// TIA Portal V19 export
FUNCTION "AUTO_LOGIC_FOR_CIP_TANK" : Void   // FC13, LAD
{ S7_Optimized_Access := 'TRUE' }
// stored: SetENOAutomatically false
   VAR_TEMP   // added for the SCL form of the ladder/FBD networks
      _w1 : Bool;
      _w2 : Bool;
      _w3 : Bool;
      _w4 : Bool;
   END_VAR
BEGIN

REGION Network 1: START
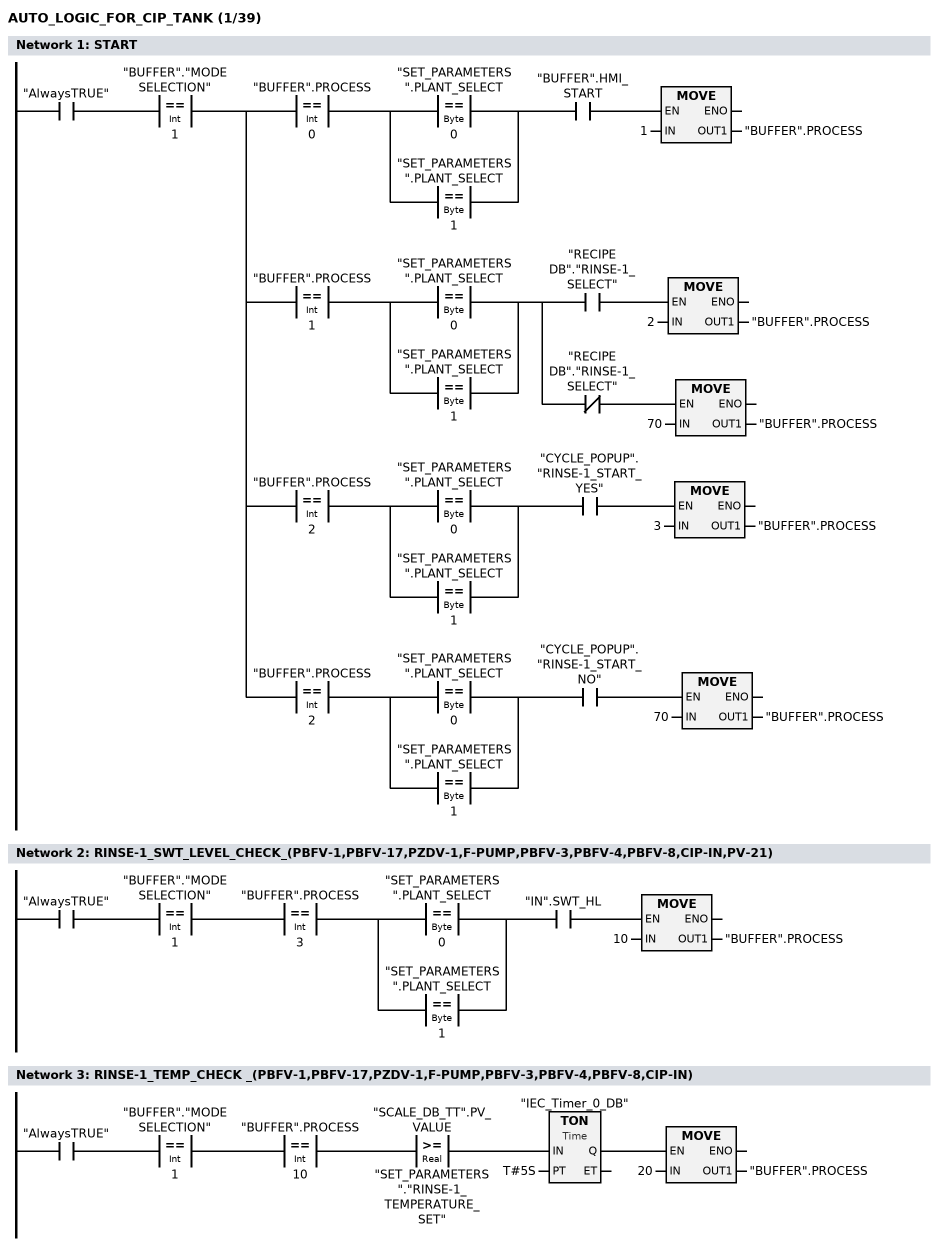
   RUNG wire#powerrail
      Contact( "AlwaysTRUE" )
      { S7_Templates := "SrcType := Int" } EQ_Contact(in1 := "BUFFER"."MODE SELECTION", in2 := 1)
      wire#w1
      { S7_Templates := "SrcType := Int" } EQ_Contact(in1 := "BUFFER".PROCESS, in2 := 0)
      wire#w2
      { S7_Templates := "SrcType := Byte" } EQ_Contact(in1 := "SET_PARAMETERS".PLANT_SELECT, in2 := 0)
      wire#w3
      Contact( "BUFFER".HMI_START )
      Move(in := 1, out1 => "BUFFER".PROCESS)
   END_RUNG
   RUNG wire#w2
      { S7_Templates := "SrcType := Byte" } EQ_Contact(in1 := "SET_PARAMETERS".PLANT_SELECT, in2 := 1)
   END_RUNG wire#w3
   RUNG wire#w1
      { S7_Templates := "SrcType := Int" } EQ_Contact(in1 := "BUFFER".PROCESS, in2 := 1)
      wire#w4
      { S7_Templates := "SrcType := Byte" } EQ_Contact(in1 := "SET_PARAMETERS".PLANT_SELECT, in2 := 0)
      wire#w5
      Contact( "RECIPE DB"."RINSE-1_SELECT" )
      Move(in := 2, out1 => "BUFFER".PROCESS)
   END_RUNG
   RUNG wire#w4
      { S7_Templates := "SrcType := Byte" } EQ_Contact(in1 := "SET_PARAMETERS".PLANT_SELECT, in2 := 1)
   END_RUNG wire#w5
   RUNG wire#w5
      I_Contact( "RECIPE DB"."RINSE-1_SELECT" )
      Move(in := 70, out1 => "BUFFER".PROCESS)
   END_RUNG
   RUNG wire#w1
      { S7_Templates := "SrcType := Int" } EQ_Contact(in1 := "BUFFER".PROCESS, in2 := 2)
      wire#w6
      { S7_Templates := "SrcType := Byte" } EQ_Contact(in1 := "SET_PARAMETERS".PLANT_SELECT, in2 := 0)
      wire#w7
      Contact( "CYCLE_POPUP"."RINSE-1_START_YES" )
      Move(in := 3, out1 => "BUFFER".PROCESS)
   END_RUNG
   RUNG wire#w6
      { S7_Templates := "SrcType := Byte" } EQ_Contact(in1 := "SET_PARAMETERS".PLANT_SELECT, in2 := 1)
   END_RUNG wire#w7
   RUNG wire#w1
      { S7_Templates := "SrcType := Int" } EQ_Contact(in1 := "BUFFER".PROCESS, in2 := 2)
      wire#w8
      { S7_Templates := "SrcType := Byte" } EQ_Contact(in1 := "SET_PARAMETERS".PLANT_SELECT, in2 := 0)
      wire#w9
      Contact( "CYCLE_POPUP"."RINSE-1_START_NO" )
      Move(in := 70, out1 => "BUFFER".PROCESS)
   END_RUNG
   RUNG wire#w8
      { S7_Templates := "SrcType := Byte" } EQ_Contact(in1 := "SET_PARAMETERS".PLANT_SELECT, in2 := 1)
   END_RUNG wire#w9
   // the same network as SCL:
   #_w1 := "AlwaysTRUE" AND ("BUFFER"."MODE SELECTION" = 1);
   IF #_w1 AND ("BUFFER".PROCESS = 0) AND (("SET_PARAMETERS".PLANT_SELECT = 0) OR ("SET_PARAMETERS".PLANT_SELECT = 1)) AND "BUFFER".HMI_START THEN
       "BUFFER".PROCESS := 1;
   END_IF;
   #_w2 := #_w1 AND ("BUFFER".PROCESS = 1) AND (("SET_PARAMETERS".PLANT_SELECT = 0) OR ("SET_PARAMETERS".PLANT_SELECT = 1));
   IF #_w2 AND "RECIPE DB"."RINSE-1_SELECT" THEN "BUFFER".PROCESS := 2; END_IF;
   IF #_w2 AND NOT "RECIPE DB"."RINSE-1_SELECT" THEN "BUFFER".PROCESS := 70; END_IF;
   IF #_w1 AND ("BUFFER".PROCESS = 2) AND (("SET_PARAMETERS".PLANT_SELECT = 0) OR ("SET_PARAMETERS".PLANT_SELECT = 1)) AND "CYCLE_POPUP"."RINSE-1_START_YES" THEN
       "BUFFER".PROCESS := 3;
   END_IF;
   IF #_w1 AND ("BUFFER".PROCESS = 2) AND (("SET_PARAMETERS".PLANT_SELECT = 0) OR ("SET_PARAMETERS".PLANT_SELECT = 1)) AND "CYCLE_POPUP"."RINSE-1_START_NO" THEN
       "BUFFER".PROCESS := 70;
   END_IF;
END_REGION

REGION Network 2: RINSE-1_SWT_LEVEL_CHECK_(PBFV-1,PBFV-17,PZDV-1,F-PUMP,PBFV-3,PBFV-4,PBFV-8,CIP-IN,PV-21)
   RUNG wire#powerrail
      Contact( "AlwaysTRUE" )
      { S7_Templates := "SrcType := Int" } EQ_Contact(in1 := "BUFFER"."MODE SELECTION", in2 := 1)
      { S7_Templates := "SrcType := Int" } EQ_Contact(in1 := "BUFFER".PROCESS, in2 := 3)
      wire#w1
      { S7_Templates := "SrcType := Byte" } EQ_Contact(in1 := "SET_PARAMETERS".PLANT_SELECT, in2 := 0)
      wire#w2
      Contact( "IN".SWT_HL )
      Move(in := 10, out1 => "BUFFER".PROCESS)
   END_RUNG
   RUNG wire#w1
      { S7_Templates := "SrcType := Byte" } EQ_Contact(in1 := "SET_PARAMETERS".PLANT_SELECT, in2 := 1)
   END_RUNG wire#w2
   // the same network as SCL:
   IF "AlwaysTRUE" AND ("BUFFER"."MODE SELECTION" = 1) AND ("BUFFER".PROCESS = 3) AND (("SET_PARAMETERS".PLANT_SELECT = 0) OR ("SET_PARAMETERS".PLANT_SELECT = 1)) AND "IN".SWT_HL THEN
       "BUFFER".PROCESS := 10;
   END_IF;
END_REGION

REGION Network 3: RINSE-1_TEMP_CHECK _(PBFV-1,PBFV-17,PZDV-1,F-PUMP,PBFV-3,PBFV-4,PBFV-8,CIP-IN)
   RUNG wire#powerrail
      Contact( "AlwaysTRUE" )
      { S7_Templates := "SrcType := Int" } EQ_Contact(in1 := "BUFFER"."MODE SELECTION", in2 := 1)
      { S7_Templates := "SrcType := Int" } EQ_Contact(in1 := "BUFFER".PROCESS, in2 := 10)
      { S7_Templates := "SrcType := Real" } GE_Contact(in1 := "SCALE_DB_TT".PV_VALUE, in2 := "SET_PARAMETERS"."RINSE-1_TEMPERATURE_SET")
      { S7_Templates := "time_type := Time" } "IEC_Timer_0_DB".TON(pt := T#5S, et =>)
      Move(in := 20, out1 => "BUFFER".PROCESS)
   END_RUNG
   // the same network as SCL:
   "IEC_Timer_0_DB".TON(IN := "AlwaysTRUE" AND ("BUFFER"."MODE SELECTION" = 1) AND ("BUFFER".PROCESS = 10) AND ("SCALE_DB_TT".PV_VALUE >= "SET_PARAMETERS"."RINSE-1_TEMPERATURE_SET"),
                        PT := T#5S);
   IF "IEC_Timer_0_DB".Q THEN "BUFFER".PROCESS := 20; END_IF;
END_REGION

REGION Network 4: RINSE-1_CLEANING_TIME_(PBFV-1,PBFV-17,PZDV-1,F-PUMP,PBFV-3,PBFV-4,PBFV-8,CIP-IN)
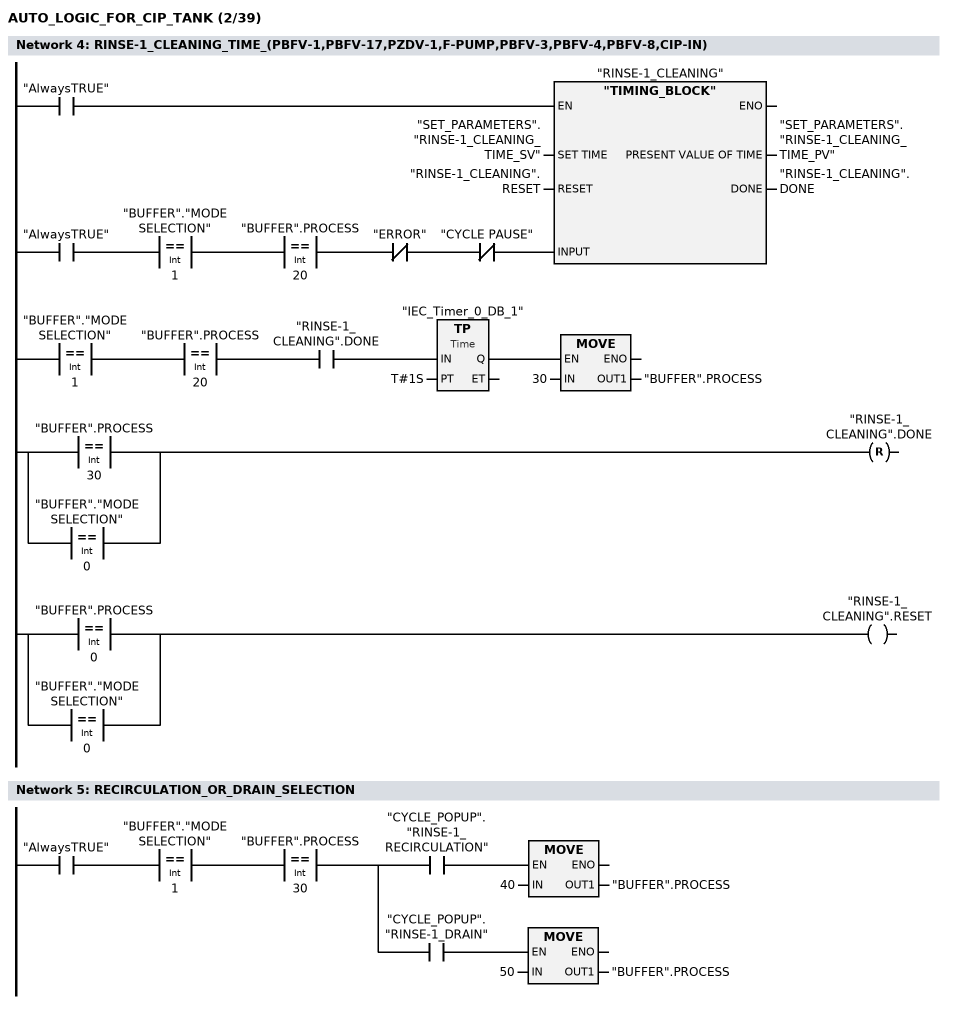
   RUNG wire#powerrail
      Contact( "AlwaysTRUE" )
      "RINSE-1_CLEANING"(INPUT := wire#w1, "SET TIME" := "SET_PARAMETERS"."RINSE-1_CLEANING_TIME_SV", RESET := "RINSE-1_CLEANING".RESET, "PRESENT VALUE OF TIME" => "SET_PARAMETERS"."RINSE-1_CLEANING_TIME_PV", DONE => "RINSE-1_CLEANING".DONE)
   END_RUNG
   RUNG wire#powerrail
      Contact( "AlwaysTRUE" )
      { S7_Templates := "SrcType := Int" } EQ_Contact(in1 := "BUFFER"."MODE SELECTION", in2 := 1)
      { S7_Templates := "SrcType := Int" } EQ_Contact(in1 := "BUFFER".PROCESS, in2 := 20)
      I_Contact( "ERROR" )
      I_Contact( "CYCLE PAUSE" )
   END_RUNG wire#w1
   RUNG wire#powerrail
      { S7_Templates := "SrcType := Int" } EQ_Contact(in1 := "BUFFER"."MODE SELECTION", in2 := 1)
      { S7_Templates := "SrcType := Int" } EQ_Contact(in1 := "BUFFER".PROCESS, in2 := 20)
      Contact( "RINSE-1_CLEANING".DONE )
      { S7_Templates := "time_type := Time" } "IEC_Timer_0_DB_1".TP(pt := T#1S, et =>)
      Move(in := 30, out1 => "BUFFER".PROCESS)
   END_RUNG
   RUNG wire#powerrail
      { S7_Templates := "SrcType := Int" } EQ_Contact(in1 := "BUFFER".PROCESS, in2 := 30)
      wire#w2
      R_Coil( "RINSE-1_CLEANING".DONE )
   END_RUNG
   RUNG wire#powerrail
      { S7_Templates := "SrcType := Int" } EQ_Contact(in1 := "BUFFER"."MODE SELECTION", in2 := 0)
   END_RUNG wire#w2
   RUNG wire#powerrail
      { S7_Templates := "SrcType := Int" } EQ_Contact(in1 := "BUFFER".PROCESS, in2 := 0)
      wire#w3
      Coil( "RINSE-1_CLEANING".RESET )
   END_RUNG
   RUNG wire#powerrail
      { S7_Templates := "SrcType := Int" } EQ_Contact(in1 := "BUFFER"."MODE SELECTION", in2 := 0)
   END_RUNG wire#w3
   // the same network as SCL:
   IF "AlwaysTRUE" THEN
       "RINSE-1_CLEANING"("SET TIME" := "SET_PARAMETERS"."RINSE-1_CLEANING_TIME_SV",   // "TIMING_BLOCK"
                          RESET := "RINSE-1_CLEANING".RESET,
                          INPUT := "AlwaysTRUE" AND ("BUFFER"."MODE SELECTION" = 1) AND ("BUFFER".PROCESS = 20) AND NOT "ERROR" AND NOT "CYCLE PAUSE",
                          "PRESENT VALUE OF TIME" => "SET_PARAMETERS"."RINSE-1_CLEANING_TIME_PV",
                          DONE => "RINSE-1_CLEANING".DONE);
   END_IF;
   "IEC_Timer_0_DB_1".TP(IN := ("BUFFER"."MODE SELECTION" = 1) AND ("BUFFER".PROCESS = 20) AND "RINSE-1_CLEANING".DONE,
                         PT := T#1S);
   IF "IEC_Timer_0_DB_1".Q THEN "BUFFER".PROCESS := 30; END_IF;
   IF ("BUFFER".PROCESS = 30) OR ("BUFFER"."MODE SELECTION" = 0) THEN
       "RINSE-1_CLEANING".DONE := FALSE;
   END_IF;
   "RINSE-1_CLEANING".RESET := ("BUFFER".PROCESS = 0) OR ("BUFFER"."MODE SELECTION" = 0);
END_REGION

REGION Network 5: RECIRCULATION_OR_DRAIN_SELECTION
   RUNG wire#powerrail
      Contact( "AlwaysTRUE" )
      { S7_Templates := "SrcType := Int" } EQ_Contact(in1 := "BUFFER"."MODE SELECTION", in2 := 1)
      { S7_Templates := "SrcType := Int" } EQ_Contact(in1 := "BUFFER".PROCESS, in2 := 30)
      wire#w1
      Contact( "CYCLE_POPUP"."RINSE-1_RECIRCULATION" )
      Move(in := 40, out1 => "BUFFER".PROCESS)
   END_RUNG
   RUNG wire#w1
      Contact( "CYCLE_POPUP"."RINSE-1_DRAIN" )
      Move(in := 50, out1 => "BUFFER".PROCESS)
   END_RUNG
   // the same network as SCL:
   #_w1 := "AlwaysTRUE" AND ("BUFFER"."MODE SELECTION" = 1) AND ("BUFFER".PROCESS = 30);
   IF #_w1 AND "CYCLE_POPUP"."RINSE-1_RECIRCULATION" THEN "BUFFER".PROCESS := 40; END_IF;
   IF #_w1 AND "CYCLE_POPUP"."RINSE-1_DRAIN" THEN "BUFFER".PROCESS := 50; END_IF;
END_REGION

REGION Network 6: RINSE-1_RECIRCULATION_TIME_(CIP-OUT,R-PUMP,PBFV-6,PBFV-8,CIP-IN)
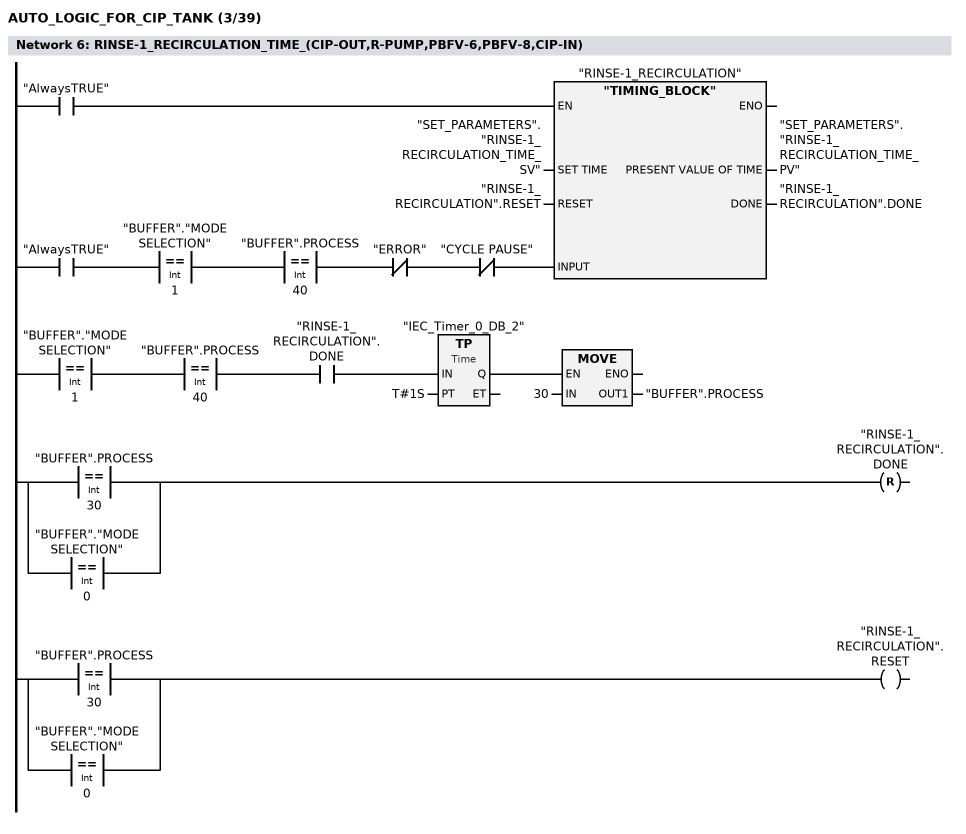
   RUNG wire#powerrail
      Contact( "AlwaysTRUE" )
      "RINSE-1_RECIRCULATION"(INPUT := wire#w1, "SET TIME" := "SET_PARAMETERS"."RINSE-1_RECIRCULATION_TIME_SV", RESET := "RINSE-1_RECIRCULATION".RESET, "PRESENT VALUE OF TIME" => "SET_PARAMETERS"."RINSE-1_RECIRCULATION_TIME_PV", DONE => "RINSE-1_RECIRCULATION".DONE)
   END_RUNG
   RUNG wire#powerrail
      Contact( "AlwaysTRUE" )
      { S7_Templates := "SrcType := Int" } EQ_Contact(in1 := "BUFFER"."MODE SELECTION", in2 := 1)
      { S7_Templates := "SrcType := Int" } EQ_Contact(in1 := "BUFFER".PROCESS, in2 := 40)
      I_Contact( "ERROR" )
      I_Contact( "CYCLE PAUSE" )
   END_RUNG wire#w1
   RUNG wire#powerrail
      { S7_Templates := "SrcType := Int" } EQ_Contact(in1 := "BUFFER"."MODE SELECTION", in2 := 1)
      { S7_Templates := "SrcType := Int" } EQ_Contact(in1 := "BUFFER".PROCESS, in2 := 40)
      Contact( "RINSE-1_RECIRCULATION".DONE )
      { S7_Templates := "time_type := Time" } "IEC_Timer_0_DB_2".TP(pt := T#1S, et =>)
      Move(in := 30, out1 => "BUFFER".PROCESS)
   END_RUNG
   RUNG wire#powerrail
      { S7_Templates := "SrcType := Int" } EQ_Contact(in1 := "BUFFER".PROCESS, in2 := 30)
      wire#w2
      R_Coil( "RINSE-1_RECIRCULATION".DONE )
   END_RUNG
   RUNG wire#powerrail
      { S7_Templates := "SrcType := Int" } EQ_Contact(in1 := "BUFFER"."MODE SELECTION", in2 := 0)
   END_RUNG wire#w2
   RUNG wire#powerrail
      { S7_Templates := "SrcType := Int" } EQ_Contact(in1 := "BUFFER".PROCESS, in2 := 30)
      wire#w3
      Coil( "RINSE-1_RECIRCULATION".RESET )
   END_RUNG
   RUNG wire#powerrail
      { S7_Templates := "SrcType := Int" } EQ_Contact(in1 := "BUFFER"."MODE SELECTION", in2 := 0)
   END_RUNG wire#w3
   // the same network as SCL:
   IF "AlwaysTRUE" THEN
       "RINSE-1_RECIRCULATION"("SET TIME" := "SET_PARAMETERS"."RINSE-1_RECIRCULATION_TIME_SV",   // "TIMING_BLOCK"
                               RESET := "RINSE-1_RECIRCULATION".RESET,
                               INPUT := "AlwaysTRUE" AND ("BUFFER"."MODE SELECTION" = 1) AND ("BUFFER".PROCESS = 40) AND NOT "ERROR" AND NOT "CYCLE PAUSE",
                               "PRESENT VALUE OF TIME" => "SET_PARAMETERS"."RINSE-1_RECIRCULATION_TIME_PV",
                               DONE => "RINSE-1_RECIRCULATION".DONE);
   END_IF;
   "IEC_Timer_0_DB_2".TP(IN := ("BUFFER"."MODE SELECTION" = 1) AND ("BUFFER".PROCESS = 40) AND "RINSE-1_RECIRCULATION".DONE,
                         PT := T#1S);
   IF "IEC_Timer_0_DB_2".Q THEN "BUFFER".PROCESS := 30; END_IF;
   IF ("BUFFER".PROCESS = 30) OR ("BUFFER"."MODE SELECTION" = 0) THEN
       "RINSE-1_RECIRCULATION".DONE := FALSE;
   END_IF;
   "RINSE-1_RECIRCULATION".RESET := ("BUFFER".PROCESS = 30) OR ("BUFFER"."MODE SELECTION" = 0);
END_REGION

REGION Network 7: RINSE-1_DRAIN_TIME_(CIP-OUT,R_PUMP,PBFV-11)
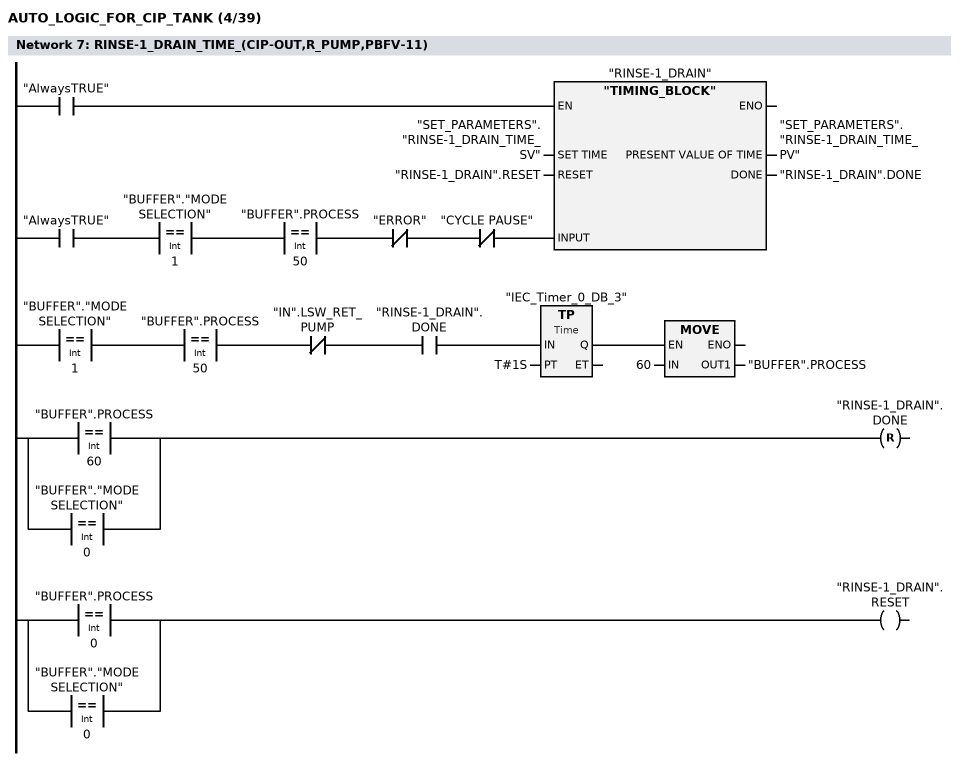
   RUNG wire#powerrail
      Contact( "AlwaysTRUE" )
      "RINSE-1_DRAIN"(INPUT := wire#w1, "SET TIME" := "SET_PARAMETERS"."RINSE-1_DRAIN_TIME_SV", RESET := "RINSE-1_DRAIN".RESET, "PRESENT VALUE OF TIME" => "SET_PARAMETERS"."RINSE-1_DRAIN_TIME_PV", DONE => "RINSE-1_DRAIN".DONE)
   END_RUNG
   RUNG wire#powerrail
      Contact( "AlwaysTRUE" )
      { S7_Templates := "SrcType := Int" } EQ_Contact(in1 := "BUFFER"."MODE SELECTION", in2 := 1)
      { S7_Templates := "SrcType := Int" } EQ_Contact(in1 := "BUFFER".PROCESS, in2 := 50)
      I_Contact( "ERROR" )
      I_Contact( "CYCLE PAUSE" )
   END_RUNG wire#w1
   RUNG wire#powerrail
      { S7_Templates := "SrcType := Int" } EQ_Contact(in1 := "BUFFER"."MODE SELECTION", in2 := 1)
      { S7_Templates := "SrcType := Int" } EQ_Contact(in1 := "BUFFER".PROCESS, in2 := 50)
      I_Contact( "IN".LSW_RET_PUMP )
      Contact( "RINSE-1_DRAIN".DONE )
      { S7_Templates := "time_type := Time" } "IEC_Timer_0_DB_3".TP(pt := T#1S, et =>)
      Move(in := 60, out1 => "BUFFER".PROCESS)
   END_RUNG
   RUNG wire#powerrail
      { S7_Templates := "SrcType := Int" } EQ_Contact(in1 := "BUFFER".PROCESS, in2 := 60)
      wire#w2
      R_Coil( "RINSE-1_DRAIN".DONE )
   END_RUNG
   RUNG wire#powerrail
      { S7_Templates := "SrcType := Int" } EQ_Contact(in1 := "BUFFER"."MODE SELECTION", in2 := 0)
   END_RUNG wire#w2
   RUNG wire#powerrail
      { S7_Templates := "SrcType := Int" } EQ_Contact(in1 := "BUFFER".PROCESS, in2 := 0)
      wire#w3
      Coil( "RINSE-1_DRAIN".RESET )
   END_RUNG
   RUNG wire#powerrail
      { S7_Templates := "SrcType := Int" } EQ_Contact(in1 := "BUFFER"."MODE SELECTION", in2 := 0)
   END_RUNG wire#w3
   // the same network as SCL:
   IF "AlwaysTRUE" THEN
       "RINSE-1_DRAIN"("SET TIME" := "SET_PARAMETERS"."RINSE-1_DRAIN_TIME_SV",   // "TIMING_BLOCK"
                       RESET := "RINSE-1_DRAIN".RESET,
                       INPUT := "AlwaysTRUE" AND ("BUFFER"."MODE SELECTION" = 1) AND ("BUFFER".PROCESS = 50) AND NOT "ERROR" AND NOT "CYCLE PAUSE",
                       "PRESENT VALUE OF TIME" => "SET_PARAMETERS"."RINSE-1_DRAIN_TIME_PV",
                       DONE => "RINSE-1_DRAIN".DONE);
   END_IF;
   "IEC_Timer_0_DB_3".TP(IN := ("BUFFER"."MODE SELECTION" = 1) AND ("BUFFER".PROCESS = 50) AND NOT "IN".LSW_RET_PUMP AND "RINSE-1_DRAIN".DONE,
                         PT := T#1S);
   IF "IEC_Timer_0_DB_3".Q THEN "BUFFER".PROCESS := 60; END_IF;
   IF ("BUFFER".PROCESS = 60) OR ("BUFFER"."MODE SELECTION" = 0) THEN "RINSE-1_DRAIN".DONE := FALSE; END_IF;
   "RINSE-1_DRAIN".RESET := ("BUFFER".PROCESS = 0) OR ("BUFFER"."MODE SELECTION" = 0);
END_REGION

REGION Network 8: RINSE-1_PUMP_CHASING_TIME(PBFV-12,PBFV13)
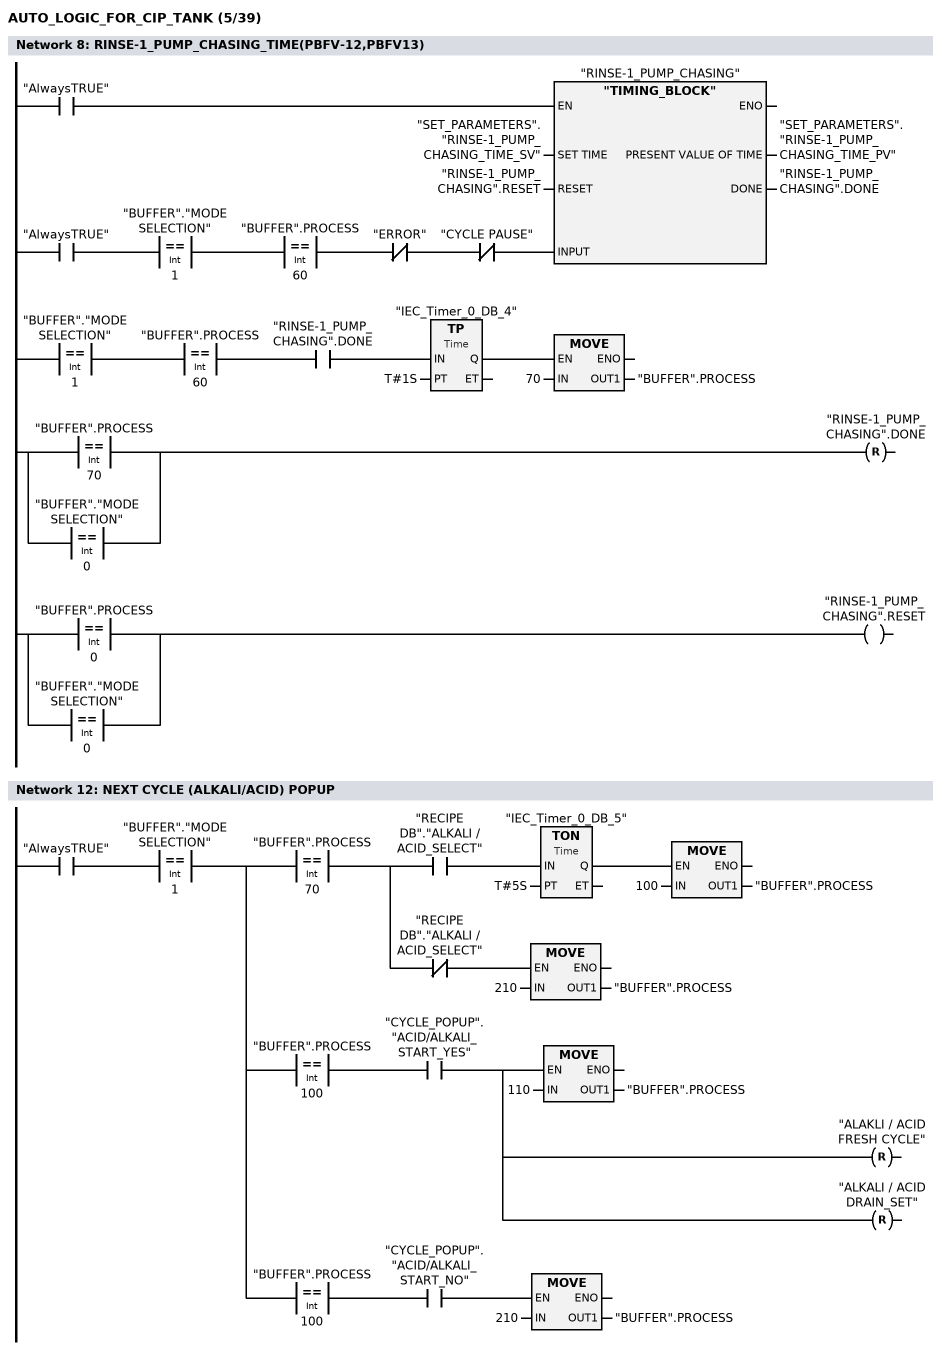
   RUNG wire#powerrail
      Contact( "AlwaysTRUE" )
      "RINSE-1_PUMP_CHASING"(INPUT := wire#w1, "SET TIME" := "SET_PARAMETERS"."RINSE-1_PUMP_CHASING_TIME_SV", RESET := "RINSE-1_PUMP_CHASING".RESET, "PRESENT VALUE OF TIME" => "SET_PARAMETERS"."RINSE-1_PUMP_CHASING_TIME_PV", DONE => "RINSE-1_PUMP_CHASING".DONE)
   END_RUNG
   RUNG wire#powerrail
      Contact( "AlwaysTRUE" )
      { S7_Templates := "SrcType := Int" } EQ_Contact(in1 := "BUFFER"."MODE SELECTION", in2 := 1)
      { S7_Templates := "SrcType := Int" } EQ_Contact(in1 := "BUFFER".PROCESS, in2 := 60)
      I_Contact( "ERROR" )
      I_Contact( "CYCLE PAUSE" )
   END_RUNG wire#w1
   RUNG wire#powerrail
      { S7_Templates := "SrcType := Int" } EQ_Contact(in1 := "BUFFER"."MODE SELECTION", in2 := 1)
      { S7_Templates := "SrcType := Int" } EQ_Contact(in1 := "BUFFER".PROCESS, in2 := 60)
      Contact( "RINSE-1_PUMP_CHASING".DONE )
      { S7_Templates := "time_type := Time" } "IEC_Timer_0_DB_4".TP(pt := T#1S, et =>)
      Move(in := 70, out1 => "BUFFER".PROCESS)
   END_RUNG
   RUNG wire#powerrail
      { S7_Templates := "SrcType := Int" } EQ_Contact(in1 := "BUFFER".PROCESS, in2 := 70)
      wire#w2
      R_Coil( "RINSE-1_PUMP_CHASING".DONE )
   END_RUNG
   RUNG wire#powerrail
      { S7_Templates := "SrcType := Int" } EQ_Contact(in1 := "BUFFER"."MODE SELECTION", in2 := 0)
   END_RUNG wire#w2
   RUNG wire#powerrail
      { S7_Templates := "SrcType := Int" } EQ_Contact(in1 := "BUFFER".PROCESS, in2 := 0)
      wire#w3
      Coil( "RINSE-1_PUMP_CHASING".RESET )
   END_RUNG
   RUNG wire#powerrail
      { S7_Templates := "SrcType := Int" } EQ_Contact(in1 := "BUFFER"."MODE SELECTION", in2 := 0)
   END_RUNG wire#w3
   // the same network as SCL:
   IF "AlwaysTRUE" THEN
       "RINSE-1_PUMP_CHASING"("SET TIME" := "SET_PARAMETERS"."RINSE-1_PUMP_CHASING_TIME_SV",   // "TIMING_BLOCK"
                              RESET := "RINSE-1_PUMP_CHASING".RESET,
                              INPUT := "AlwaysTRUE" AND ("BUFFER"."MODE SELECTION" = 1) AND ("BUFFER".PROCESS = 60) AND NOT "ERROR" AND NOT "CYCLE PAUSE",
                              "PRESENT VALUE OF TIME" => "SET_PARAMETERS"."RINSE-1_PUMP_CHASING_TIME_PV",
                              DONE => "RINSE-1_PUMP_CHASING".DONE);
   END_IF;
   "IEC_Timer_0_DB_4".TP(IN := ("BUFFER"."MODE SELECTION" = 1) AND ("BUFFER".PROCESS = 60) AND "RINSE-1_PUMP_CHASING".DONE,
                         PT := T#1S);
   IF "IEC_Timer_0_DB_4".Q THEN "BUFFER".PROCESS := 70; END_IF;
   IF ("BUFFER".PROCESS = 70) OR ("BUFFER"."MODE SELECTION" = 0) THEN
       "RINSE-1_PUMP_CHASING".DONE := FALSE;
   END_IF;
   "RINSE-1_PUMP_CHASING".RESET := ("BUFFER".PROCESS = 0) OR ("BUFFER"."MODE SELECTION" = 0);
END_REGION

REGION Network 12: NEXT CYCLE (ALKALI/ACID) POPUP
   RUNG wire#powerrail
      Contact( "AlwaysTRUE" )
      { S7_Templates := "SrcType := Int" } EQ_Contact(in1 := "BUFFER"."MODE SELECTION", in2 := 1)
      wire#w1
      { S7_Templates := "SrcType := Int" } EQ_Contact(in1 := "BUFFER".PROCESS, in2 := 70)
      wire#w2
      Contact( "RECIPE DB"."ALKALI / ACID_SELECT" )
      { S7_Templates := "time_type := Time" } "IEC_Timer_0_DB_5".TON(pt := T#5S, et =>)
      Move(in := 100, out1 => "BUFFER".PROCESS)
   END_RUNG
   RUNG wire#w2
      I_Contact( "RECIPE DB"."ALKALI / ACID_SELECT" )
      Move(in := 210, out1 => "BUFFER".PROCESS)
   END_RUNG
   RUNG wire#w1
      { S7_Templates := "SrcType := Int" } EQ_Contact(in1 := "BUFFER".PROCESS, in2 := 100)
      Contact( "CYCLE_POPUP"."ACID/ALKALI_START_YES" )
      wire#w3
      Move(in := 110, out1 => "BUFFER".PROCESS)
   END_RUNG
   RUNG wire#w3
      R_Coil( "ALAKLI / ACID FRESH CYCLE" )
   END_RUNG
   RUNG wire#w3
      R_Coil( "ALKALI / ACID DRAIN_SET" )
   END_RUNG
   RUNG wire#w1
      { S7_Templates := "SrcType := Int" } EQ_Contact(in1 := "BUFFER".PROCESS, in2 := 100)
      Contact( "CYCLE_POPUP"."ACID/ALKALI_START_NO" )
      Move(in := 210, out1 => "BUFFER".PROCESS)
   END_RUNG
   // the same network as SCL:
   #_w1 := "AlwaysTRUE" AND ("BUFFER"."MODE SELECTION" = 1);
   #_w2 := #_w1 AND ("BUFFER".PROCESS = 70);
   "IEC_Timer_0_DB_5".TON(IN := #_w2 AND "RECIPE DB"."ALKALI / ACID_SELECT", PT := T#5S);
   IF "IEC_Timer_0_DB_5".Q THEN "BUFFER".PROCESS := 100; END_IF;
   IF #_w2 AND NOT "RECIPE DB"."ALKALI / ACID_SELECT" THEN "BUFFER".PROCESS := 210; END_IF;
   #_w3 := #_w1 AND ("BUFFER".PROCESS = 100) AND "CYCLE_POPUP"."ACID/ALKALI_START_YES";
   IF #_w3 THEN
       "BUFFER".PROCESS := 110;
       "ALAKLI / ACID FRESH CYCLE" := FALSE;
       "ALKALI / ACID DRAIN_SET" := FALSE;
   END_IF;
   IF #_w1 AND ("BUFFER".PROCESS = 100) AND "CYCLE_POPUP"."ACID/ALKALI_START_NO" THEN
       "BUFFER".PROCESS := 210;
   END_IF;
END_REGION

REGION Network 13: SWT_LEVEL_CHECK(PBFV-17) POPUP + temperature cleaing
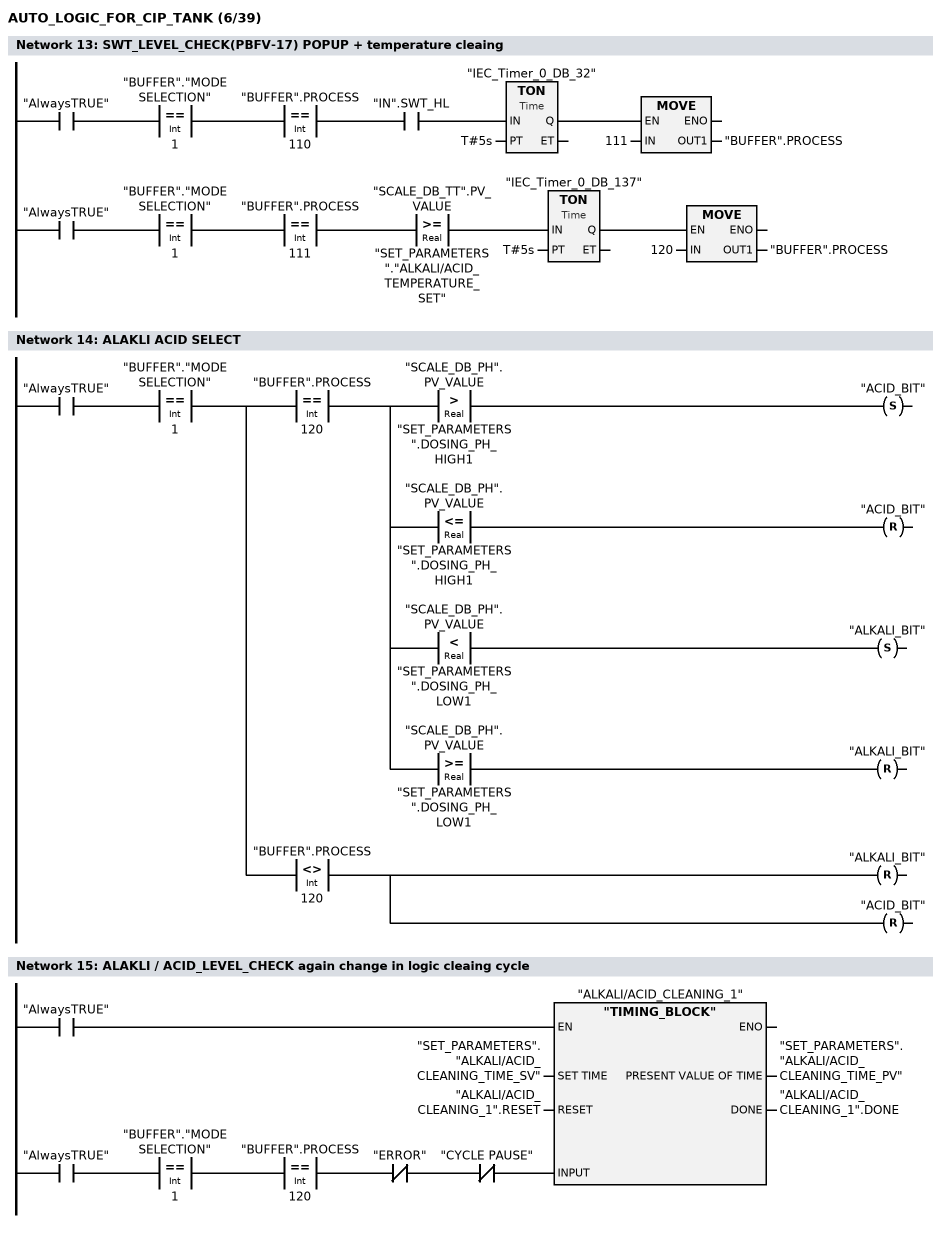
   RUNG wire#powerrail
      Contact( "AlwaysTRUE" )
      { S7_Templates := "SrcType := Int" } EQ_Contact(in1 := "BUFFER"."MODE SELECTION", in2 := 1)
      { S7_Templates := "SrcType := Int" } EQ_Contact(in1 := "BUFFER".PROCESS, in2 := 110)
      Contact( "IN".SWT_HL )
      { S7_Templates := "time_type := Time" } "IEC_Timer_0_DB_32".TON(pt := T#5s, et =>)
      Move(in := 111, out1 => "BUFFER".PROCESS)
   END_RUNG
   RUNG wire#powerrail
      Contact( "AlwaysTRUE" )
      { S7_Templates := "SrcType := Int" } EQ_Contact(in1 := "BUFFER"."MODE SELECTION", in2 := 1)
      { S7_Templates := "SrcType := Int" } EQ_Contact(in1 := "BUFFER".PROCESS, in2 := 111)
      { S7_Templates := "SrcType := Real" } GE_Contact(in1 := "SCALE_DB_TT".PV_VALUE, in2 := "SET_PARAMETERS"."ALKALI/ACID_TEMPERATURE_SET")
      { S7_Templates := "time_type := Time" } "IEC_Timer_0_DB_137".TON(pt := T#5s, et =>)
      Move(in := 120, out1 => "BUFFER".PROCESS)
   END_RUNG
   // the same network as SCL:
   "IEC_Timer_0_DB_32".TON(IN := "AlwaysTRUE" AND ("BUFFER"."MODE SELECTION" = 1) AND ("BUFFER".PROCESS = 110) AND "IN".SWT_HL,
                           PT := T#5s);
   IF "IEC_Timer_0_DB_32".Q THEN "BUFFER".PROCESS := 111; END_IF;
   "IEC_Timer_0_DB_137".TON(IN := "AlwaysTRUE" AND ("BUFFER"."MODE SELECTION" = 1) AND ("BUFFER".PROCESS = 111) AND ("SCALE_DB_TT".PV_VALUE >= "SET_PARAMETERS"."ALKALI/ACID_TEMPERATURE_SET"),
                           PT := T#5s);
   IF "IEC_Timer_0_DB_137".Q THEN "BUFFER".PROCESS := 120; END_IF;
END_REGION

REGION Network 14: ALAKLI ACID SELECT
   RUNG wire#powerrail
      Contact( "AlwaysTRUE" )
      { S7_Templates := "SrcType := Int" } EQ_Contact(in1 := "BUFFER"."MODE SELECTION", in2 := 1)
      wire#w1
      { S7_Templates := "SrcType := Int" } EQ_Contact(in1 := "BUFFER".PROCESS, in2 := 120)
      wire#w2
      { S7_Templates := "SrcType := Real" } GT_Contact(in1 := "SCALE_DB_PH".PV_VALUE, in2 := "SET_PARAMETERS".DOSING_PH_HIGH1)
      S_Coil( "ACID_BIT" )
   END_RUNG
   RUNG wire#w2
      { S7_Templates := "SrcType := Real" } LE_Contact(in1 := "SCALE_DB_PH".PV_VALUE, in2 := "SET_PARAMETERS".DOSING_PH_HIGH1)
      R_Coil( "ACID_BIT" )
   END_RUNG
   RUNG wire#w2
      { S7_Templates := "SrcType := Real" } LT_Contact(in1 := "SCALE_DB_PH".PV_VALUE, in2 := "SET_PARAMETERS".DOSING_PH_LOW1)
      S_Coil( "ALKALI_BIT" )
   END_RUNG
   RUNG wire#w2
      { S7_Templates := "SrcType := Real" } GE_Contact(in1 := "SCALE_DB_PH".PV_VALUE, in2 := "SET_PARAMETERS".DOSING_PH_LOW1)
      R_Coil( "ALKALI_BIT" )
   END_RUNG
   RUNG wire#w1
      { S7_Templates := "SrcType := Int" } NE_Contact(in1 := "BUFFER".PROCESS, in2 := 120)
      wire#w3
      R_Coil( "ALKALI_BIT" )
   END_RUNG
   RUNG wire#w3
      R_Coil( "ACID_BIT" )
   END_RUNG
   // the same network as SCL:
   #_w1 := "AlwaysTRUE" AND ("BUFFER"."MODE SELECTION" = 1);
   #_w2 := #_w1 AND ("BUFFER".PROCESS = 120);
   IF #_w2 AND ("SCALE_DB_PH".PV_VALUE > "SET_PARAMETERS".DOSING_PH_HIGH1) THEN "ACID_BIT" := TRUE; END_IF;
   IF #_w2 AND ("SCALE_DB_PH".PV_VALUE <= "SET_PARAMETERS".DOSING_PH_HIGH1) THEN "ACID_BIT" := FALSE; END_IF;
   IF #_w2 AND ("SCALE_DB_PH".PV_VALUE < "SET_PARAMETERS".DOSING_PH_LOW1) THEN "ALKALI_BIT" := TRUE; END_IF;
   IF #_w2 AND ("SCALE_DB_PH".PV_VALUE >= "SET_PARAMETERS".DOSING_PH_LOW1) THEN
       "ALKALI_BIT" := FALSE;
   END_IF;
   IF #_w1 AND ("BUFFER".PROCESS <> 120) THEN
       "ALKALI_BIT" := FALSE;
       "ACID_BIT" := FALSE;
   END_IF;
END_REGION

REGION Network 15: ALAKLI / ACID_LEVEL_CHECK again change in logic cleaing cycle
   RUNG wire#powerrail
      Contact( "AlwaysTRUE" )
      "ALKALI/ACID_CLEANING_1"(INPUT := wire#w1, "SET TIME" := "SET_PARAMETERS"."ALKALI/ACID_CLEANING_TIME_SV", RESET := "ALKALI/ACID_CLEANING_1".RESET, "PRESENT VALUE OF TIME" => "SET_PARAMETERS"."ALKALI/ACID_CLEANING_TIME_PV", DONE => "ALKALI/ACID_CLEANING_1".DONE)
   END_RUNG
   RUNG wire#powerrail
      Contact( "AlwaysTRUE" )
      { S7_Templates := "SrcType := Int" } EQ_Contact(in1 := "BUFFER"."MODE SELECTION", in2 := 1)
      { S7_Templates := "SrcType := Int" } EQ_Contact(in1 := "BUFFER".PROCESS, in2 := 120)
      I_Contact( "ERROR" )
      I_Contact( "CYCLE PAUSE" )
   END_RUNG wire#w1
   // the same network as SCL:
   IF "AlwaysTRUE" THEN
       "ALKALI/ACID_CLEANING_1"("SET TIME" := "SET_PARAMETERS"."ALKALI/ACID_CLEANING_TIME_SV",   // "TIMING_BLOCK"
                               RESET := "ALKALI/ACID_CLEANING_1".RESET,
                               INPUT := "AlwaysTRUE" AND ("BUFFER"."MODE SELECTION" = 1) AND ("BUFFER".PROCESS = 120) AND NOT "ERROR" AND NOT "CYCLE PAUSE",
                               "PRESENT VALUE OF TIME" => "SET_PARAMETERS"."ALKALI/ACID_CLEANING_TIME_PV",
                               DONE => "ALKALI/ACID_CLEANING_1".DONE);
   END_IF;
END_REGION

REGION Network 16: use------------------
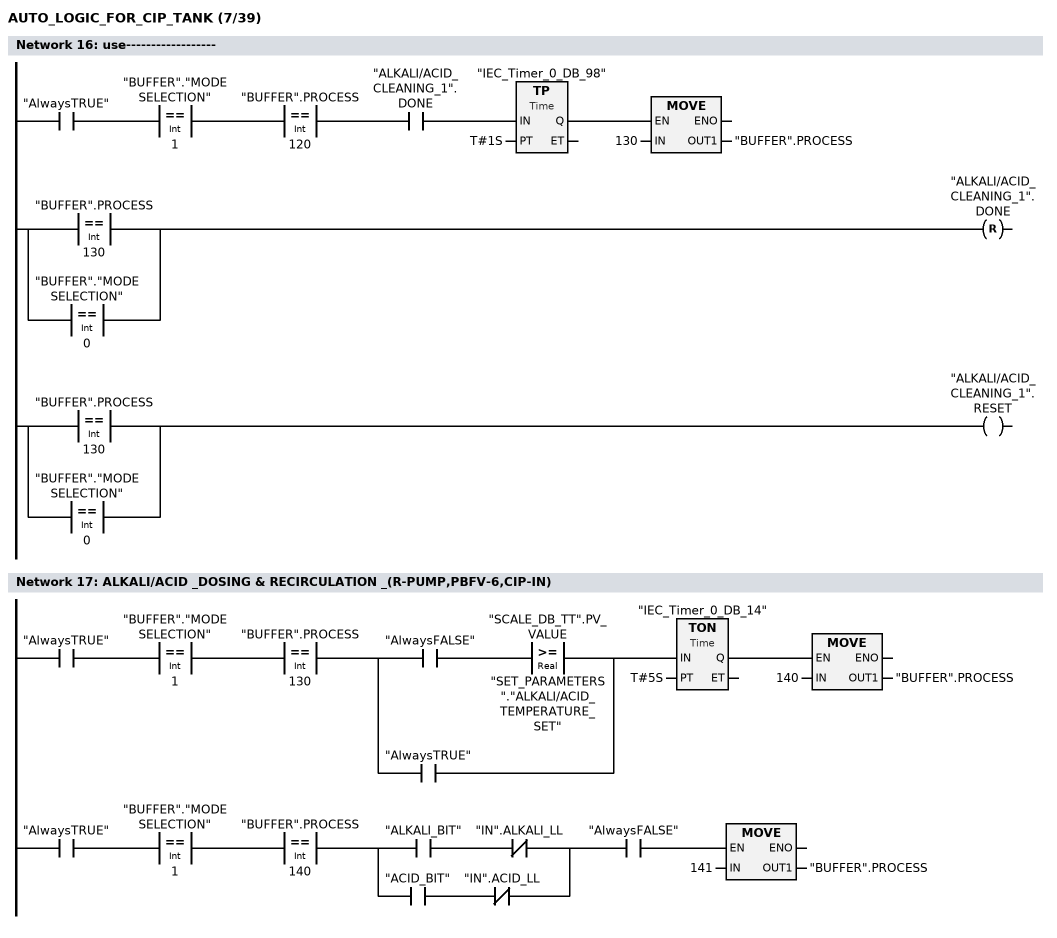
   RUNG wire#powerrail
      Contact( "AlwaysTRUE" )
      { S7_Templates := "SrcType := Int" } EQ_Contact(in1 := "BUFFER"."MODE SELECTION", in2 := 1)
      { S7_Templates := "SrcType := Int" } EQ_Contact(in1 := "BUFFER".PROCESS, in2 := 120)
      Contact( "ALKALI/ACID_CLEANING_1".DONE )
      { S7_Templates := "time_type := Time" } "IEC_Timer_0_DB_98".TP(pt := T#1S, et =>)
      Move(in := 130, out1 => "BUFFER".PROCESS)
   END_RUNG
   RUNG wire#powerrail
      { S7_Templates := "SrcType := Int" } EQ_Contact(in1 := "BUFFER".PROCESS, in2 := 130)
      wire#w1
      R_Coil( "ALKALI/ACID_CLEANING_1".DONE )
   END_RUNG
   RUNG wire#powerrail
      { S7_Templates := "SrcType := Int" } EQ_Contact(in1 := "BUFFER"."MODE SELECTION", in2 := 0)
   END_RUNG wire#w1
   RUNG wire#powerrail
      { S7_Templates := "SrcType := Int" } EQ_Contact(in1 := "BUFFER".PROCESS, in2 := 130)
      wire#w2
      Coil( "ALKALI/ACID_CLEANING_1".RESET )
   END_RUNG
   RUNG wire#powerrail
      { S7_Templates := "SrcType := Int" } EQ_Contact(in1 := "BUFFER"."MODE SELECTION", in2 := 0)
   END_RUNG wire#w2
   // the same network as SCL:
   "IEC_Timer_0_DB_98".TP(IN := "AlwaysTRUE" AND ("BUFFER"."MODE SELECTION" = 1) AND ("BUFFER".PROCESS = 120) AND "ALKALI/ACID_CLEANING_1".DONE,
                          PT := T#1S);
   IF "IEC_Timer_0_DB_98".Q THEN "BUFFER".PROCESS := 130; END_IF;
   IF ("BUFFER".PROCESS = 130) OR ("BUFFER"."MODE SELECTION" = 0) THEN
       "ALKALI/ACID_CLEANING_1".DONE := FALSE;
   END_IF;
   "ALKALI/ACID_CLEANING_1".RESET := ("BUFFER".PROCESS = 130) OR ("BUFFER"."MODE SELECTION" = 0);
END_REGION

REGION Network 17: ALKALI/ACID _DOSING & RECIRCULATION _(R-PUMP,PBFV-6,CIP-IN)
   RUNG wire#powerrail
      Contact( "AlwaysTRUE" )
      { S7_Templates := "SrcType := Int" } EQ_Contact(in1 := "BUFFER"."MODE SELECTION", in2 := 1)
      { S7_Templates := "SrcType := Int" } EQ_Contact(in1 := "BUFFER".PROCESS, in2 := 130)
      wire#w1
      Contact( "AlwaysFALSE" )
      { S7_Templates := "SrcType := Real" } GE_Contact(in1 := "SCALE_DB_TT".PV_VALUE, in2 := "SET_PARAMETERS"."ALKALI/ACID_TEMPERATURE_SET")
      wire#w2
      { S7_Templates := "time_type := Time" } "IEC_Timer_0_DB_14".TON(pt := T#5S, et =>)
      Move(in := 140, out1 => "BUFFER".PROCESS)
   END_RUNG
   RUNG wire#w1
      Contact( "AlwaysTRUE" )
   END_RUNG wire#w2
   RUNG wire#powerrail
      Contact( "AlwaysTRUE" )
      { S7_Templates := "SrcType := Int" } EQ_Contact(in1 := "BUFFER"."MODE SELECTION", in2 := 1)
      { S7_Templates := "SrcType := Int" } EQ_Contact(in1 := "BUFFER".PROCESS, in2 := 140)
      wire#w3
      Contact( "ALKALI_BIT" )
      I_Contact( "IN".ALKALI_LL )
      wire#w4
      Contact( "AlwaysFALSE" )
      Move(in := 141, out1 => "BUFFER".PROCESS)
   END_RUNG
   RUNG wire#w3
      Contact( "ACID_BIT" )
      I_Contact( "IN".ACID_LL )
   END_RUNG wire#w4
   // the same network as SCL:
   "IEC_Timer_0_DB_14".TON(IN := "AlwaysTRUE" AND ("BUFFER"."MODE SELECTION" = 1) AND ("BUFFER".PROCESS = 130) AND (("AlwaysFALSE" AND ("SCALE_DB_TT".PV_VALUE >= "SET_PARAMETERS"."ALKALI/ACID_TEMPERATURE_SET")) OR "AlwaysTRUE"),
                           PT := T#5S);
   IF "IEC_Timer_0_DB_14".Q THEN "BUFFER".PROCESS := 140; END_IF;
   IF "AlwaysTRUE" AND ("BUFFER"."MODE SELECTION" = 1) AND ("BUFFER".PROCESS = 140) AND (("ALKALI_BIT" AND NOT "IN".ALKALI_LL) OR ("ACID_BIT" AND NOT "IN".ACID_LL)) AND "AlwaysFALSE" THEN
       "BUFFER".PROCESS := 141;
   END_IF;
END_REGION

REGION Network 18: ALKALI/ACID_RECIRCULATION_TIME_(CIP-OUT,R-PUMP,PBFV-6,PBFV-8,CIP-IN)
   // recirculation + dosing
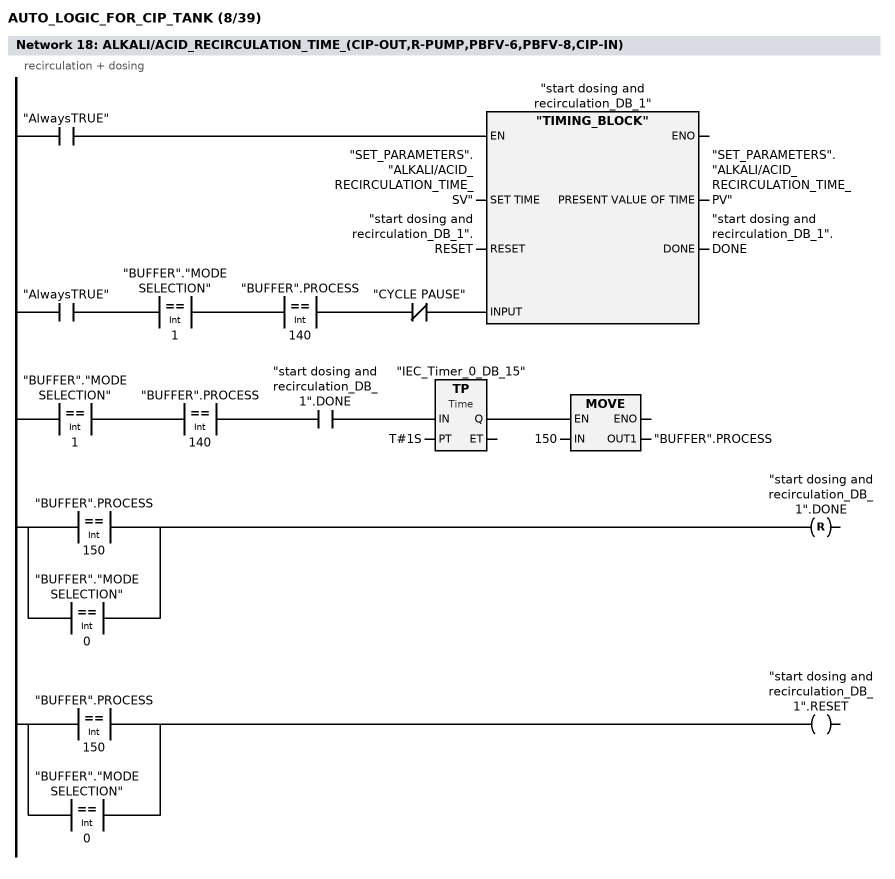
   RUNG wire#powerrail
      Contact( "AlwaysTRUE" )
      "start dosing and recirculation_DB_1"(INPUT := wire#w1, "SET TIME" := "SET_PARAMETERS"."ALKALI/ACID_RECIRCULATION_TIME_SV", RESET := "start dosing and recirculation_DB_1".RESET, "PRESENT VALUE OF TIME" => "SET_PARAMETERS"."ALKALI/ACID_RECIRCULATION_TIME_PV", DONE => "start dosing and recirculation_DB_1".DONE)
   END_RUNG
   RUNG wire#powerrail
      Contact( "AlwaysTRUE" )
      { S7_Templates := "SrcType := Int" } EQ_Contact(in1 := "BUFFER"."MODE SELECTION", in2 := 1)
      { S7_Templates := "SrcType := Int" } EQ_Contact(in1 := "BUFFER".PROCESS, in2 := 140)
      I_Contact( "CYCLE PAUSE" )
   END_RUNG wire#w1
   RUNG wire#powerrail
      { S7_Templates := "SrcType := Int" } EQ_Contact(in1 := "BUFFER"."MODE SELECTION", in2 := 1)
      { S7_Templates := "SrcType := Int" } EQ_Contact(in1 := "BUFFER".PROCESS, in2 := 140)
      Contact( "start dosing and recirculation_DB_1".DONE )
      { S7_Templates := "time_type := Time" } "IEC_Timer_0_DB_15".TP(pt := T#1S, et =>)
      Move(in := 150, out1 => "BUFFER".PROCESS)
   END_RUNG
   RUNG wire#powerrail
      { S7_Templates := "SrcType := Int" } EQ_Contact(in1 := "BUFFER".PROCESS, in2 := 150)
      wire#w2
      R_Coil( "start dosing and recirculation_DB_1".DONE )
   END_RUNG
   RUNG wire#powerrail
      { S7_Templates := "SrcType := Int" } EQ_Contact(in1 := "BUFFER"."MODE SELECTION", in2 := 0)
   END_RUNG wire#w2
   RUNG wire#powerrail
      { S7_Templates := "SrcType := Int" } EQ_Contact(in1 := "BUFFER".PROCESS, in2 := 150)
      wire#w3
      Coil( "start dosing and recirculation_DB_1".RESET )
   END_RUNG
   RUNG wire#powerrail
      { S7_Templates := "SrcType := Int" } EQ_Contact(in1 := "BUFFER"."MODE SELECTION", in2 := 0)
   END_RUNG wire#w3
   // the same network as SCL:
   IF "AlwaysTRUE" THEN
       "start dosing and recirculation_DB_1"("SET TIME" := "SET_PARAMETERS"."ALKALI/ACID_RECIRCULATION_TIME_SV",   // "TIMING_BLOCK"
                               RESET := "start dosing and recirculation_DB_1".RESET,
                               INPUT := "AlwaysTRUE" AND ("BUFFER"."MODE SELECTION" = 1) AND ("BUFFER".PROCESS = 140) AND NOT "CYCLE PAUSE",
                               "PRESENT VALUE OF TIME" => "SET_PARAMETERS"."ALKALI/ACID_RECIRCULATION_TIME_PV",
                               DONE => "start dosing and recirculation_DB_1".DONE);
   END_IF;
   "IEC_Timer_0_DB_15".TP(IN := ("BUFFER"."MODE SELECTION" = 1) AND ("BUFFER".PROCESS = 140) AND "start dosing and recirculation_DB_1".DONE,
                          PT := T#1S);
   IF "IEC_Timer_0_DB_15".Q THEN "BUFFER".PROCESS := 150; END_IF;
   IF ("BUFFER".PROCESS = 150) OR ("BUFFER"."MODE SELECTION" = 0) THEN
       "start dosing and recirculation_DB_1".DONE := FALSE;
   END_IF;
   "start dosing and recirculation_DB_1".RESET := ("BUFFER".PROCESS = 150) OR ("BUFFER"."MODE SELECTION" = 0);
END_REGION

REGION Network 19: PH ACHIEVED OR NOT ACHIEVED BIT SET FOR POPUP.
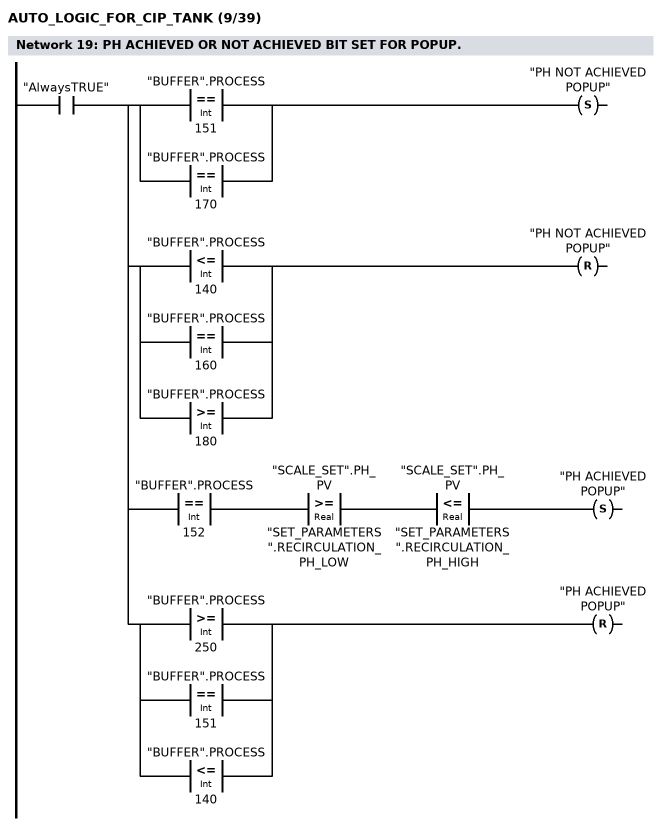
   RUNG wire#powerrail
      Contact( "AlwaysTRUE" )
      wire#w1
      { S7_Templates := "SrcType := Int" } EQ_Contact(in1 := "BUFFER".PROCESS, in2 := 151)
      wire#w2
      S_Coil( "PH NOT ACHIEVED POPUP" )
   END_RUNG
   RUNG wire#w1
      { S7_Templates := "SrcType := Int" } EQ_Contact(in1 := "BUFFER".PROCESS, in2 := 170)
   END_RUNG wire#w2
   RUNG wire#w1
      { S7_Templates := "SrcType := Int" } LE_Contact(in1 := "BUFFER".PROCESS, in2 := 140)
      wire#w3
      R_Coil( "PH NOT ACHIEVED POPUP" )
   END_RUNG
   RUNG wire#w1
      { S7_Templates := "SrcType := Int" } EQ_Contact(in1 := "BUFFER".PROCESS, in2 := 160)
   END_RUNG wire#w3
   RUNG wire#w1
      { S7_Templates := "SrcType := Int" } GE_Contact(in1 := "BUFFER".PROCESS, in2 := 180)
   END_RUNG wire#w3
   RUNG wire#w1
      { S7_Templates := "SrcType := Int" } EQ_Contact(in1 := "BUFFER".PROCESS, in2 := 152)
      { S7_Templates := "SrcType := Real" } GE_Contact(in1 := "SCALE_SET".PH_PV, in2 := "SET_PARAMETERS".RECIRCULATION_PH_LOW)
      { S7_Templates := "SrcType := Real" } LE_Contact(in1 := "SCALE_SET".PH_PV, in2 := "SET_PARAMETERS".RECIRCULATION_PH_HIGH)
      S_Coil( "PH ACHIEVED POPUP" )
   END_RUNG
   RUNG wire#w1
      { S7_Templates := "SrcType := Int" } GE_Contact(in1 := "BUFFER".PROCESS, in2 := 250)
      wire#w4
      R_Coil( "PH ACHIEVED POPUP" )
   END_RUNG
   RUNG wire#w1
      { S7_Templates := "SrcType := Int" } EQ_Contact(in1 := "BUFFER".PROCESS, in2 := 151)
   END_RUNG wire#w4
   RUNG wire#w1
      { S7_Templates := "SrcType := Int" } LE_Contact(in1 := "BUFFER".PROCESS, in2 := 140)
   END_RUNG wire#w4
   // the same network as SCL:
   IF "AlwaysTRUE" AND (("BUFFER".PROCESS = 151) OR ("BUFFER".PROCESS = 170)) THEN
       "PH NOT ACHIEVED POPUP" := TRUE;
   END_IF;
   IF "AlwaysTRUE" AND (("BUFFER".PROCESS <= 140) OR ("BUFFER".PROCESS = 160) OR ("BUFFER".PROCESS >= 180)) THEN
       "PH NOT ACHIEVED POPUP" := FALSE;
   END_IF;
   IF "AlwaysTRUE" AND ("BUFFER".PROCESS = 152) AND ("SCALE_SET".PH_PV >= "SET_PARAMETERS".RECIRCULATION_PH_LOW) AND ("SCALE_SET".PH_PV <= "SET_PARAMETERS".RECIRCULATION_PH_HIGH) THEN
       "PH ACHIEVED POPUP" := TRUE;
   END_IF;
   IF "AlwaysTRUE" AND (("BUFFER".PROCESS >= 250) OR ("BUFFER".PROCESS = 151) OR ("BUFFER".PROCESS <= 140)) THEN
       "PH ACHIEVED POPUP" := FALSE;
   END_IF;
END_REGION

REGION Network 20: ALKALI/ACID_PH CHECKING_TIME_
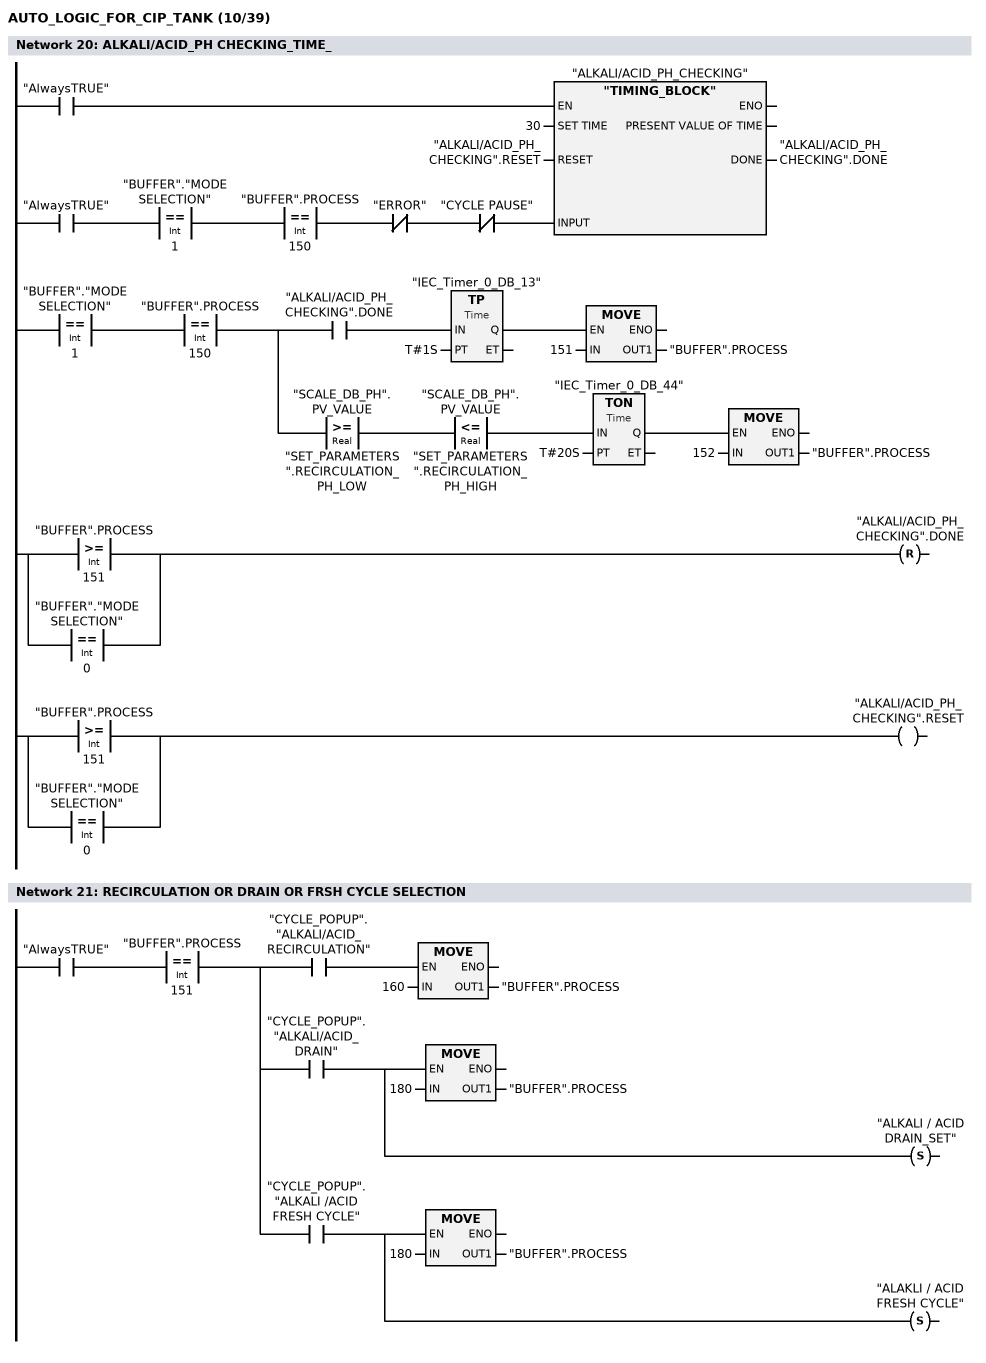
   RUNG wire#powerrail
      Contact( "AlwaysTRUE" )
      "ALKALI/ACID_PH_CHECKING"(INPUT := wire#w1, "SET TIME" := 30, RESET := "ALKALI/ACID_PH_CHECKING".RESET, "PRESENT VALUE OF TIME" =>, DONE => "ALKALI/ACID_PH_CHECKING".DONE)
   END_RUNG
   RUNG wire#powerrail
      Contact( "AlwaysTRUE" )
      { S7_Templates := "SrcType := Int" } EQ_Contact(in1 := "BUFFER"."MODE SELECTION", in2 := 1)
      { S7_Templates := "SrcType := Int" } EQ_Contact(in1 := "BUFFER".PROCESS, in2 := 150)
      I_Contact( "ERROR" )
      I_Contact( "CYCLE PAUSE" )
   END_RUNG wire#w1
   RUNG wire#powerrail
      { S7_Templates := "SrcType := Int" } EQ_Contact(in1 := "BUFFER"."MODE SELECTION", in2 := 1)
      { S7_Templates := "SrcType := Int" } EQ_Contact(in1 := "BUFFER".PROCESS, in2 := 150)
      wire#w2
      Contact( "ALKALI/ACID_PH_CHECKING".DONE )
      { S7_Templates := "time_type := Time" } "IEC_Timer_0_DB_13".TP(pt := T#1S, et =>)
      Move(in := 151, out1 => "BUFFER".PROCESS)
   END_RUNG
   RUNG wire#w2
      { S7_Templates := "SrcType := Real" } GE_Contact(in1 := "SCALE_DB_PH".PV_VALUE, in2 := "SET_PARAMETERS".RECIRCULATION_PH_LOW)
      { S7_Templates := "SrcType := Real" } LE_Contact(in1 := "SCALE_DB_PH".PV_VALUE, in2 := "SET_PARAMETERS".RECIRCULATION_PH_HIGH)
      { S7_Templates := "time_type := Time" } "IEC_Timer_0_DB_44".TON(pt := T#20S, et =>)
      Move(in := 152, out1 => "BUFFER".PROCESS)
   END_RUNG
   RUNG wire#powerrail
      { S7_Templates := "SrcType := Int" } GE_Contact(in1 := "BUFFER".PROCESS, in2 := 151)
      wire#w3
      R_Coil( "ALKALI/ACID_PH_CHECKING".DONE )
   END_RUNG
   RUNG wire#powerrail
      { S7_Templates := "SrcType := Int" } EQ_Contact(in1 := "BUFFER"."MODE SELECTION", in2 := 0)
   END_RUNG wire#w3
   RUNG wire#powerrail
      { S7_Templates := "SrcType := Int" } GE_Contact(in1 := "BUFFER".PROCESS, in2 := 151)
      wire#w4
      Coil( "ALKALI/ACID_PH_CHECKING".RESET )
   END_RUNG
   RUNG wire#powerrail
      { S7_Templates := "SrcType := Int" } EQ_Contact(in1 := "BUFFER"."MODE SELECTION", in2 := 0)
   END_RUNG wire#w4
   // the same network as SCL:
   IF "AlwaysTRUE" THEN
       "ALKALI/ACID_PH_CHECKING"("SET TIME" := 30,   // "TIMING_BLOCK"
                               RESET := "ALKALI/ACID_PH_CHECKING".RESET,
                               INPUT := "AlwaysTRUE" AND ("BUFFER"."MODE SELECTION" = 1) AND ("BUFFER".PROCESS = 150) AND NOT "ERROR" AND NOT "CYCLE PAUSE",
                               DONE => "ALKALI/ACID_PH_CHECKING".DONE);
   END_IF;
   #_w1 := ("BUFFER"."MODE SELECTION" = 1) AND ("BUFFER".PROCESS = 150);
   "IEC_Timer_0_DB_13".TP(IN := #_w1 AND "ALKALI/ACID_PH_CHECKING".DONE, PT := T#1S);
   IF "IEC_Timer_0_DB_13".Q THEN "BUFFER".PROCESS := 151; END_IF;
   "IEC_Timer_0_DB_44".TON(IN := #_w1 AND ("SCALE_DB_PH".PV_VALUE >= "SET_PARAMETERS".RECIRCULATION_PH_LOW) AND ("SCALE_DB_PH".PV_VALUE <= "SET_PARAMETERS".RECIRCULATION_PH_HIGH),
                           PT := T#20S);
   IF "IEC_Timer_0_DB_44".Q THEN "BUFFER".PROCESS := 152; END_IF;
   IF ("BUFFER".PROCESS >= 151) OR ("BUFFER"."MODE SELECTION" = 0) THEN
       "ALKALI/ACID_PH_CHECKING".DONE := FALSE;
   END_IF;
   "ALKALI/ACID_PH_CHECKING".RESET := ("BUFFER".PROCESS >= 151) OR ("BUFFER"."MODE SELECTION" = 0);
END_REGION

REGION Network 21: RECIRCULATION OR DRAIN OR FRSH CYCLE SELECTION
   RUNG wire#powerrail
      Contact( "AlwaysTRUE" )
      { S7_Templates := "SrcType := Int" } EQ_Contact(in1 := "BUFFER".PROCESS, in2 := 151)
      wire#w1
      Contact( "CYCLE_POPUP"."ALKALI/ACID_RECIRCULATION" )
      Move(in := 160, out1 => "BUFFER".PROCESS)
   END_RUNG
   RUNG wire#w1
      Contact( "CYCLE_POPUP"."ALKALI/ACID_DRAIN" )
      wire#w2
      Move(in := 180, out1 => "BUFFER".PROCESS)
   END_RUNG
   RUNG wire#w2
      S_Coil( "ALKALI / ACID DRAIN_SET" )
   END_RUNG
   RUNG wire#w1
      Contact( "CYCLE_POPUP"."ALKALI /ACID FRESH CYCLE" )
      wire#w3
      Move(in := 180, out1 => "BUFFER".PROCESS)
   END_RUNG
   RUNG wire#w3
      S_Coil( "ALAKLI / ACID FRESH CYCLE" )
   END_RUNG
   // the same network as SCL:
   #_w1 := "AlwaysTRUE" AND ("BUFFER".PROCESS = 151);
   IF #_w1 AND "CYCLE_POPUP"."ALKALI/ACID_RECIRCULATION" THEN "BUFFER".PROCESS := 160; END_IF;
   IF #_w1 AND "CYCLE_POPUP"."ALKALI/ACID_DRAIN" THEN
       "BUFFER".PROCESS := 180;
       "ALKALI / ACID DRAIN_SET" := TRUE;
   END_IF;
   IF #_w1 AND "CYCLE_POPUP"."ALKALI /ACID FRESH CYCLE" THEN
       "BUFFER".PROCESS := 180;
       "ALAKLI / ACID FRESH CYCLE" := TRUE;
   END_IF;
END_REGION

REGION Network 22: PH ACHIEVED GONG TO DRAIN
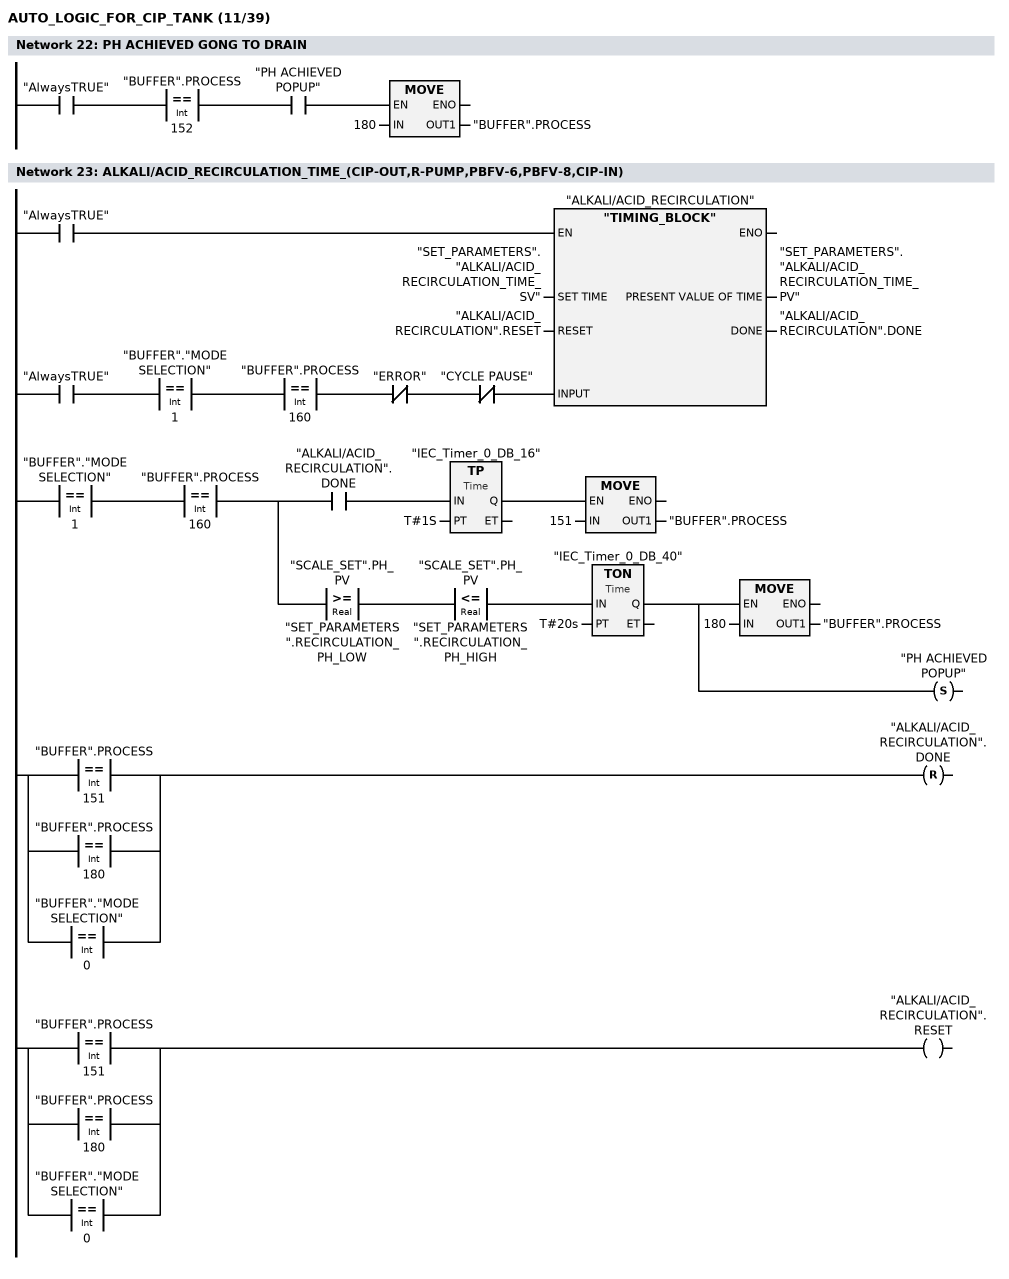
   RUNG wire#powerrail
      Contact( "AlwaysTRUE" )
      { S7_Templates := "SrcType := Int" } EQ_Contact(in1 := "BUFFER".PROCESS, in2 := 152)
      Contact( "PH ACHIEVED POPUP" )
      Move(in := 180, out1 => "BUFFER".PROCESS)
   END_RUNG
   // the same network as SCL:
   IF "AlwaysTRUE" AND ("BUFFER".PROCESS = 152) AND "PH ACHIEVED POPUP" THEN "BUFFER".PROCESS := 180; END_IF;
END_REGION

REGION Network 23: ALKALI/ACID_RECIRCULATION_TIME_(CIP-OUT,R-PUMP,PBFV-6,PBFV-8,CIP-IN)
   RUNG wire#powerrail
      Contact( "AlwaysTRUE" )
      "ALKALI/ACID_RECIRCULATION"(INPUT := wire#w1, "SET TIME" := "SET_PARAMETERS"."ALKALI/ACID_RECIRCULATION_TIME_SV", RESET := "ALKALI/ACID_RECIRCULATION".RESET, "PRESENT VALUE OF TIME" => "SET_PARAMETERS"."ALKALI/ACID_RECIRCULATION_TIME_PV", DONE => "ALKALI/ACID_RECIRCULATION".DONE)
   END_RUNG
   RUNG wire#powerrail
      Contact( "AlwaysTRUE" )
      { S7_Templates := "SrcType := Int" } EQ_Contact(in1 := "BUFFER"."MODE SELECTION", in2 := 1)
      { S7_Templates := "SrcType := Int" } EQ_Contact(in1 := "BUFFER".PROCESS, in2 := 160)
      I_Contact( "ERROR" )
      I_Contact( "CYCLE PAUSE" )
   END_RUNG wire#w1
   RUNG wire#powerrail
      { S7_Templates := "SrcType := Int" } EQ_Contact(in1 := "BUFFER"."MODE SELECTION", in2 := 1)
      { S7_Templates := "SrcType := Int" } EQ_Contact(in1 := "BUFFER".PROCESS, in2 := 160)
      wire#w2
      Contact( "ALKALI/ACID_RECIRCULATION".DONE )
      { S7_Templates := "time_type := Time" } "IEC_Timer_0_DB_16".TP(pt := T#1S, et =>)
      Move(in := 151, out1 => "BUFFER".PROCESS)
   END_RUNG
   RUNG wire#w2
      { S7_Templates := "SrcType := Real" } GE_Contact(in1 := "SCALE_SET".PH_PV, in2 := "SET_PARAMETERS".RECIRCULATION_PH_LOW)
      { S7_Templates := "SrcType := Real" } LE_Contact(in1 := "SCALE_SET".PH_PV, in2 := "SET_PARAMETERS".RECIRCULATION_PH_HIGH)
      { S7_Templates := "time_type := Time" } "IEC_Timer_0_DB_40".TON(pt := T#20s, et =>)
      wire#w3
      Move(in := 180, out1 => "BUFFER".PROCESS)
   END_RUNG
   RUNG wire#w3
      S_Coil( "PH ACHIEVED POPUP" )
   END_RUNG
   RUNG wire#powerrail
      { S7_Templates := "SrcType := Int" } EQ_Contact(in1 := "BUFFER".PROCESS, in2 := 151)
      wire#w4
      R_Coil( "ALKALI/ACID_RECIRCULATION".DONE )
   END_RUNG
   RUNG wire#powerrail
      { S7_Templates := "SrcType := Int" } EQ_Contact(in1 := "BUFFER".PROCESS, in2 := 180)
   END_RUNG wire#w4
   RUNG wire#powerrail
      { S7_Templates := "SrcType := Int" } EQ_Contact(in1 := "BUFFER"."MODE SELECTION", in2 := 0)
   END_RUNG wire#w4
   RUNG wire#powerrail
      { S7_Templates := "SrcType := Int" } EQ_Contact(in1 := "BUFFER".PROCESS, in2 := 151)
      wire#w5
      Coil( "ALKALI/ACID_RECIRCULATION".RESET )
   END_RUNG
   RUNG wire#powerrail
      { S7_Templates := "SrcType := Int" } EQ_Contact(in1 := "BUFFER".PROCESS, in2 := 180)
   END_RUNG wire#w5
   RUNG wire#powerrail
      { S7_Templates := "SrcType := Int" } EQ_Contact(in1 := "BUFFER"."MODE SELECTION", in2 := 0)
   END_RUNG wire#w5
   // the same network as SCL:
   IF "AlwaysTRUE" THEN
       "ALKALI/ACID_RECIRCULATION"("SET TIME" := "SET_PARAMETERS"."ALKALI/ACID_RECIRCULATION_TIME_SV",   // "TIMING_BLOCK"
                               RESET := "ALKALI/ACID_RECIRCULATION".RESET,
                               INPUT := "AlwaysTRUE" AND ("BUFFER"."MODE SELECTION" = 1) AND ("BUFFER".PROCESS = 160) AND NOT "ERROR" AND NOT "CYCLE PAUSE",
                               "PRESENT VALUE OF TIME" => "SET_PARAMETERS"."ALKALI/ACID_RECIRCULATION_TIME_PV",
                               DONE => "ALKALI/ACID_RECIRCULATION".DONE);
   END_IF;
   #_w1 := ("BUFFER"."MODE SELECTION" = 1) AND ("BUFFER".PROCESS = 160);
   "IEC_Timer_0_DB_16".TP(IN := #_w1 AND "ALKALI/ACID_RECIRCULATION".DONE, PT := T#1S);
   IF "IEC_Timer_0_DB_16".Q THEN "BUFFER".PROCESS := 151; END_IF;
   "IEC_Timer_0_DB_40".TON(IN := #_w1 AND ("SCALE_SET".PH_PV >= "SET_PARAMETERS".RECIRCULATION_PH_LOW) AND ("SCALE_SET".PH_PV <= "SET_PARAMETERS".RECIRCULATION_PH_HIGH),
                           PT := T#20s);
   IF "IEC_Timer_0_DB_40".Q THEN
       "BUFFER".PROCESS := 180;
       "PH ACHIEVED POPUP" := TRUE;
   END_IF;
   IF ("BUFFER".PROCESS = 151) OR ("BUFFER".PROCESS = 180) OR ("BUFFER"."MODE SELECTION" = 0) THEN
       "ALKALI/ACID_RECIRCULATION".DONE := FALSE;
   END_IF;
   "ALKALI/ACID_RECIRCULATION".RESET := ("BUFFER".PROCESS = 151) OR ("BUFFER".PROCESS = 180) OR ("BUFFER"."MODE SELECTION" = 0);
END_REGION

REGION Network 24: ALKALI/ACID_DRAIN_TIME_(CIP-OUT,R_PUMP,PBFV-11)
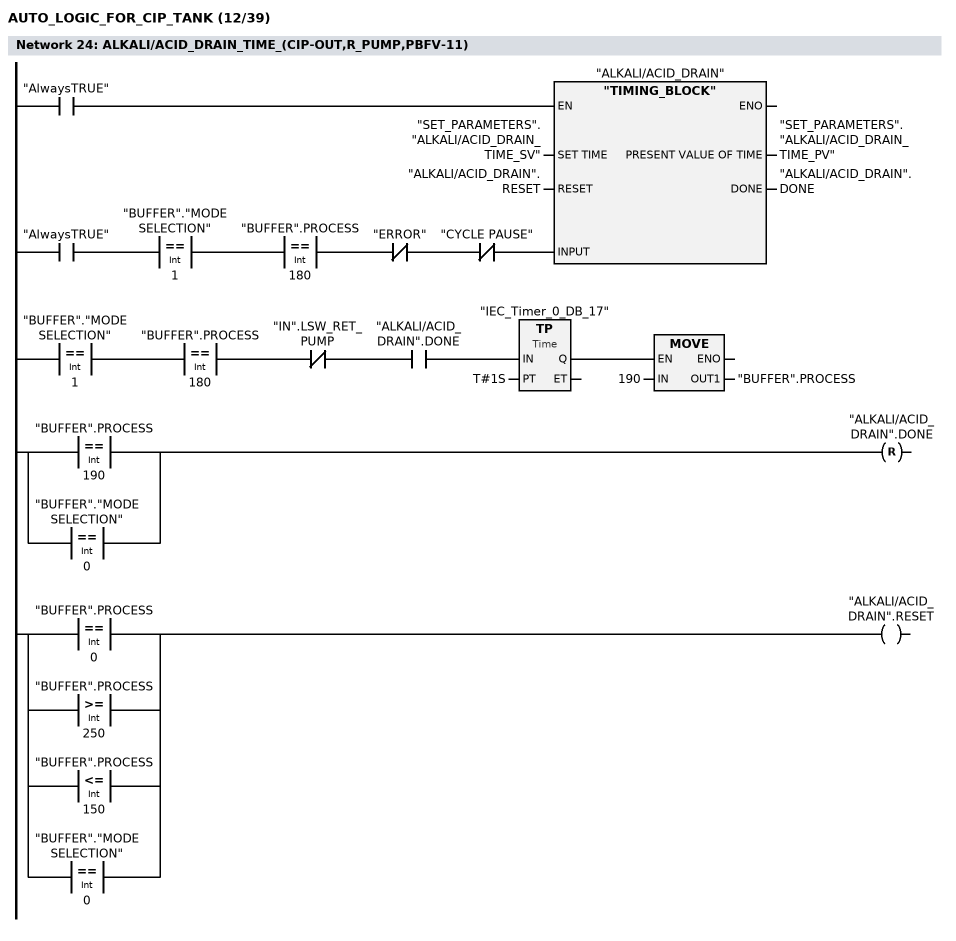
   RUNG wire#powerrail
      Contact( "AlwaysTRUE" )
      "ALKALI/ACID_DRAIN"(INPUT := wire#w1, "SET TIME" := "SET_PARAMETERS"."ALKALI/ACID_DRAIN_TIME_SV", RESET := "ALKALI/ACID_DRAIN".RESET, "PRESENT VALUE OF TIME" => "SET_PARAMETERS"."ALKALI/ACID_DRAIN_TIME_PV", DONE => "ALKALI/ACID_DRAIN".DONE)
   END_RUNG
   RUNG wire#powerrail
      Contact( "AlwaysTRUE" )
      { S7_Templates := "SrcType := Int" } EQ_Contact(in1 := "BUFFER"."MODE SELECTION", in2 := 1)
      { S7_Templates := "SrcType := Int" } EQ_Contact(in1 := "BUFFER".PROCESS, in2 := 180)
      I_Contact( "ERROR" )
      I_Contact( "CYCLE PAUSE" )
   END_RUNG wire#w1
   RUNG wire#powerrail
      { S7_Templates := "SrcType := Int" } EQ_Contact(in1 := "BUFFER"."MODE SELECTION", in2 := 1)
      { S7_Templates := "SrcType := Int" } EQ_Contact(in1 := "BUFFER".PROCESS, in2 := 180)
      I_Contact( "IN".LSW_RET_PUMP )
      Contact( "ALKALI/ACID_DRAIN".DONE )
      { S7_Templates := "time_type := Time" } "IEC_Timer_0_DB_17".TP(pt := T#1S, et =>)
      Move(in := 190, out1 => "BUFFER".PROCESS)
   END_RUNG
   RUNG wire#powerrail
      { S7_Templates := "SrcType := Int" } EQ_Contact(in1 := "BUFFER".PROCESS, in2 := 190)
      wire#w2
      R_Coil( "ALKALI/ACID_DRAIN".DONE )
   END_RUNG
   RUNG wire#powerrail
      { S7_Templates := "SrcType := Int" } EQ_Contact(in1 := "BUFFER"."MODE SELECTION", in2 := 0)
   END_RUNG wire#w2
   RUNG wire#powerrail
      { S7_Templates := "SrcType := Int" } EQ_Contact(in1 := "BUFFER".PROCESS, in2 := 0)
      wire#w3
      Coil( "ALKALI/ACID_DRAIN".RESET )
   END_RUNG
   RUNG wire#powerrail
      { S7_Templates := "SrcType := Int" } GE_Contact(in1 := "BUFFER".PROCESS, in2 := 250)
   END_RUNG wire#w3
   RUNG wire#powerrail
      { S7_Templates := "SrcType := Int" } LE_Contact(in1 := "BUFFER".PROCESS, in2 := 150)
   END_RUNG wire#w3
   RUNG wire#powerrail
      { S7_Templates := "SrcType := Int" } EQ_Contact(in1 := "BUFFER"."MODE SELECTION", in2 := 0)
   END_RUNG wire#w3
   // the same network as SCL:
   IF "AlwaysTRUE" THEN
       "ALKALI/ACID_DRAIN"("SET TIME" := "SET_PARAMETERS"."ALKALI/ACID_DRAIN_TIME_SV",   // "TIMING_BLOCK"
                           RESET := "ALKALI/ACID_DRAIN".RESET,
                           INPUT := "AlwaysTRUE" AND ("BUFFER"."MODE SELECTION" = 1) AND ("BUFFER".PROCESS = 180) AND NOT "ERROR" AND NOT "CYCLE PAUSE",
                           "PRESENT VALUE OF TIME" => "SET_PARAMETERS"."ALKALI/ACID_DRAIN_TIME_PV",
                           DONE => "ALKALI/ACID_DRAIN".DONE);
   END_IF;
   "IEC_Timer_0_DB_17".TP(IN := ("BUFFER"."MODE SELECTION" = 1) AND ("BUFFER".PROCESS = 180) AND NOT "IN".LSW_RET_PUMP AND "ALKALI/ACID_DRAIN".DONE,
                          PT := T#1S);
   IF "IEC_Timer_0_DB_17".Q THEN "BUFFER".PROCESS := 190; END_IF;
   IF ("BUFFER".PROCESS = 190) OR ("BUFFER"."MODE SELECTION" = 0) THEN
       "ALKALI/ACID_DRAIN".DONE := FALSE;
   END_IF;
   "ALKALI/ACID_DRAIN".RESET := ("BUFFER".PROCESS = 0) OR ("BUFFER".PROCESS >= 250) OR ("BUFFER".PROCESS <= 150) OR ("BUFFER"."MODE SELECTION" = 0);
END_REGION

REGION Network 25: ALKALI/ACID_PUMP_CHASING_TIME_(PBFV-12,PBFV13)
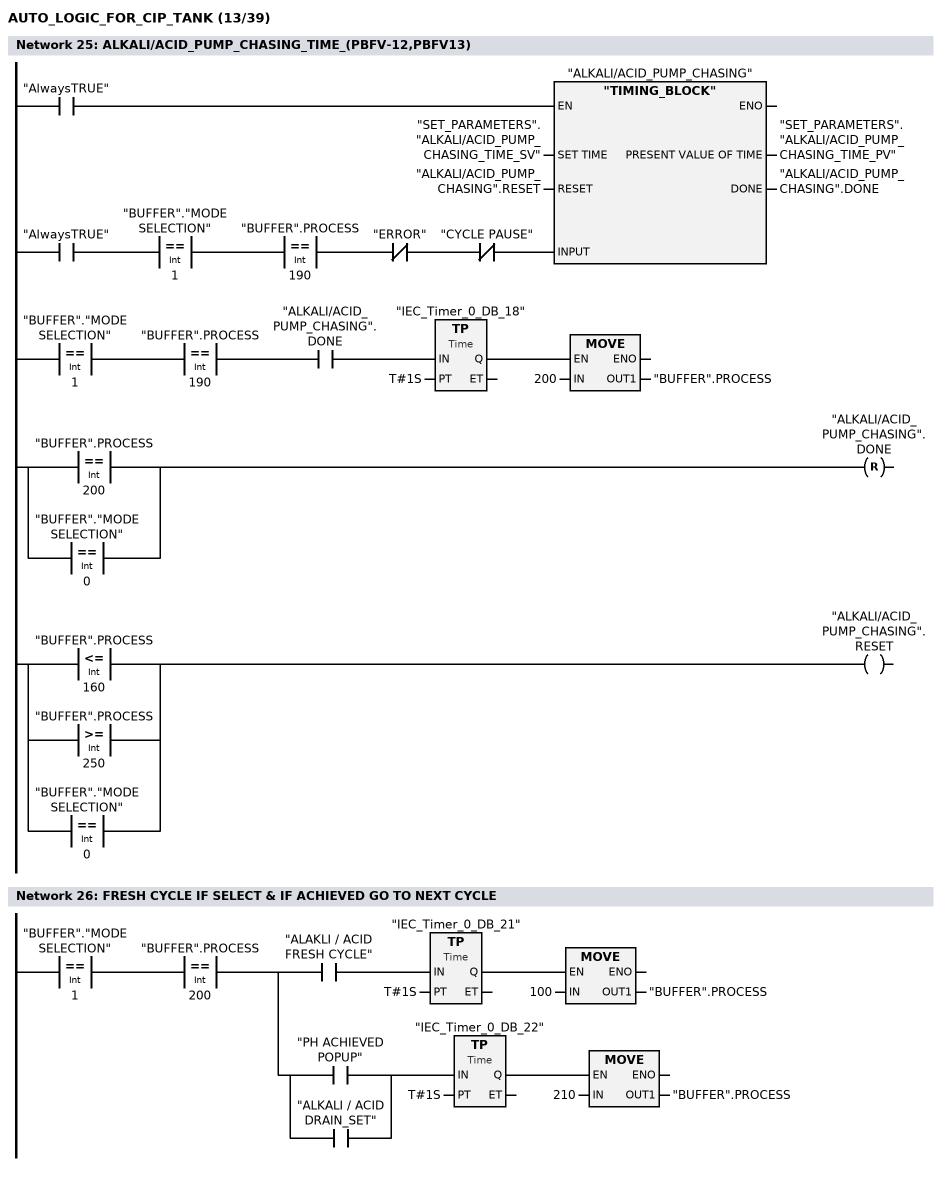
   RUNG wire#powerrail
      Contact( "AlwaysTRUE" )
      "ALKALI/ACID_PUMP_CHASING"(INPUT := wire#w1, "SET TIME" := "SET_PARAMETERS"."ALKALI/ACID_PUMP_CHASING_TIME_SV", RESET := "ALKALI/ACID_PUMP_CHASING".RESET, "PRESENT VALUE OF TIME" => "SET_PARAMETERS"."ALKALI/ACID_PUMP_CHASING_TIME_PV", DONE => "ALKALI/ACID_PUMP_CHASING".DONE)
   END_RUNG
   RUNG wire#powerrail
      Contact( "AlwaysTRUE" )
      { S7_Templates := "SrcType := Int" } EQ_Contact(in1 := "BUFFER"."MODE SELECTION", in2 := 1)
      { S7_Templates := "SrcType := Int" } EQ_Contact(in1 := "BUFFER".PROCESS, in2 := 190)
      I_Contact( "ERROR" )
      I_Contact( "CYCLE PAUSE" )
   END_RUNG wire#w1
   RUNG wire#powerrail
      { S7_Templates := "SrcType := Int" } EQ_Contact(in1 := "BUFFER"."MODE SELECTION", in2 := 1)
      { S7_Templates := "SrcType := Int" } EQ_Contact(in1 := "BUFFER".PROCESS, in2 := 190)
      Contact( "ALKALI/ACID_PUMP_CHASING".DONE )
      { S7_Templates := "time_type := Time" } "IEC_Timer_0_DB_18".TP(pt := T#1S, et =>)
      Move(in := 200, out1 => "BUFFER".PROCESS)
   END_RUNG
   RUNG wire#powerrail
      { S7_Templates := "SrcType := Int" } EQ_Contact(in1 := "BUFFER".PROCESS, in2 := 200)
      wire#w2
      R_Coil( "ALKALI/ACID_PUMP_CHASING".DONE )
   END_RUNG
   RUNG wire#powerrail
      { S7_Templates := "SrcType := Int" } EQ_Contact(in1 := "BUFFER"."MODE SELECTION", in2 := 0)
   END_RUNG wire#w2
   RUNG wire#powerrail
      { S7_Templates := "SrcType := Int" } LE_Contact(in1 := "BUFFER".PROCESS, in2 := 160)
      wire#w3
      Coil( "ALKALI/ACID_PUMP_CHASING".RESET )
   END_RUNG
   RUNG wire#powerrail
      { S7_Templates := "SrcType := Int" } GE_Contact(in1 := "BUFFER".PROCESS, in2 := 250)
   END_RUNG wire#w3
   RUNG wire#powerrail
      { S7_Templates := "SrcType := Int" } EQ_Contact(in1 := "BUFFER"."MODE SELECTION", in2 := 0)
   END_RUNG wire#w3
   // the same network as SCL:
   IF "AlwaysTRUE" THEN
       "ALKALI/ACID_PUMP_CHASING"("SET TIME" := "SET_PARAMETERS"."ALKALI/ACID_PUMP_CHASING_TIME_SV",   // "TIMING_BLOCK"
                               RESET := "ALKALI/ACID_PUMP_CHASING".RESET,
                               INPUT := "AlwaysTRUE" AND ("BUFFER"."MODE SELECTION" = 1) AND ("BUFFER".PROCESS = 190) AND NOT "ERROR" AND NOT "CYCLE PAUSE",
                               "PRESENT VALUE OF TIME" => "SET_PARAMETERS"."ALKALI/ACID_PUMP_CHASING_TIME_PV",
                               DONE => "ALKALI/ACID_PUMP_CHASING".DONE);
   END_IF;
   "IEC_Timer_0_DB_18".TP(IN := ("BUFFER"."MODE SELECTION" = 1) AND ("BUFFER".PROCESS = 190) AND "ALKALI/ACID_PUMP_CHASING".DONE,
                          PT := T#1S);
   IF "IEC_Timer_0_DB_18".Q THEN "BUFFER".PROCESS := 200; END_IF;
   IF ("BUFFER".PROCESS = 200) OR ("BUFFER"."MODE SELECTION" = 0) THEN
       "ALKALI/ACID_PUMP_CHASING".DONE := FALSE;
   END_IF;
   "ALKALI/ACID_PUMP_CHASING".RESET := ("BUFFER".PROCESS <= 160) OR ("BUFFER".PROCESS >= 250) OR ("BUFFER"."MODE SELECTION" = 0);
END_REGION

REGION Network 26: FRESH CYCLE IF SELECT & IF ACHIEVED GO TO NEXT CYCLE
   RUNG wire#powerrail
      { S7_Templates := "SrcType := Int" } EQ_Contact(in1 := "BUFFER"."MODE SELECTION", in2 := 1)
      { S7_Templates := "SrcType := Int" } EQ_Contact(in1 := "BUFFER".PROCESS, in2 := 200)
      wire#w1
      Contact( "ALAKLI / ACID FRESH CYCLE" )
      { S7_Templates := "time_type := Time" } "IEC_Timer_0_DB_21".TP(pt := T#1S, et =>)
      Move(in := 100, out1 => "BUFFER".PROCESS)
   END_RUNG
   RUNG wire#w1
      Contact( "PH ACHIEVED POPUP" )
      wire#w2
      { S7_Templates := "time_type := Time" } "IEC_Timer_0_DB_22".TP(pt := T#1S, et =>)
      Move(in := 210, out1 => "BUFFER".PROCESS)
   END_RUNG
   RUNG wire#w1
      Contact( "ALKALI / ACID DRAIN_SET" )
   END_RUNG wire#w2
   // the same network as SCL:
   #_w1 := ("BUFFER"."MODE SELECTION" = 1) AND ("BUFFER".PROCESS = 200);
   "IEC_Timer_0_DB_21".TP(IN := #_w1 AND "ALAKLI / ACID FRESH CYCLE", PT := T#1S);
   IF "IEC_Timer_0_DB_21".Q THEN "BUFFER".PROCESS := 100; END_IF;
   "IEC_Timer_0_DB_22".TP(IN := #_w1 AND ("PH ACHIEVED POPUP" OR "ALKALI / ACID DRAIN_SET"), PT := T#1S);
   IF "IEC_Timer_0_DB_22".Q THEN "BUFFER".PROCESS := 210; END_IF;
END_REGION

REGION Network 30: NEXT_CYCLE(RINSE-2) POPUP
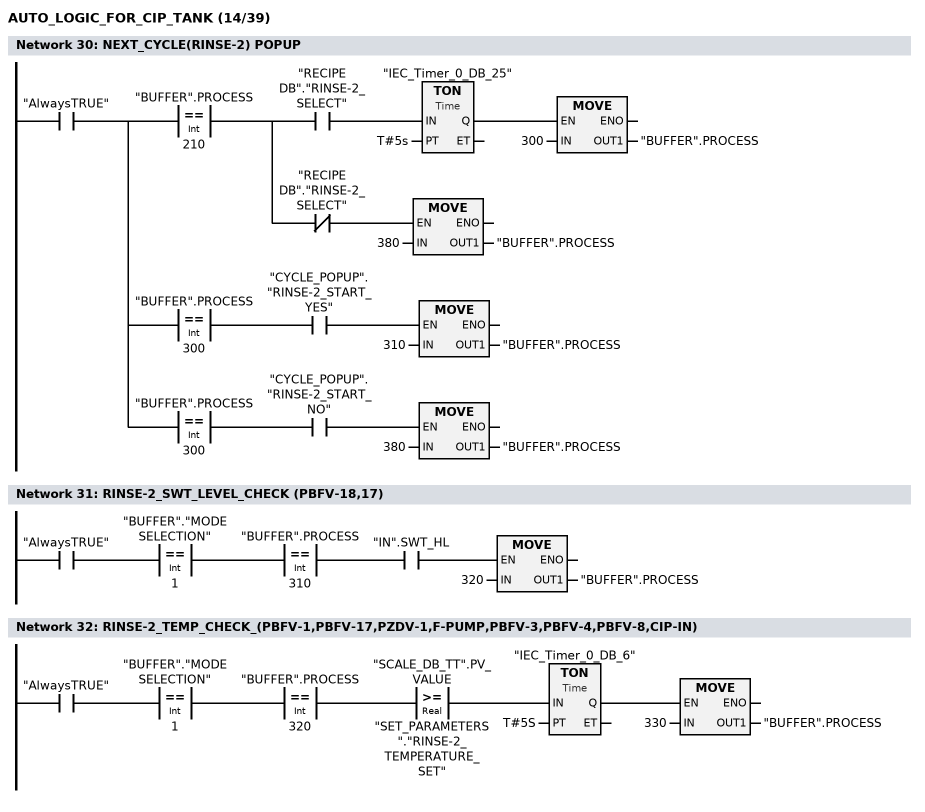
   RUNG wire#powerrail
      Contact( "AlwaysTRUE" )
      wire#w1
      { S7_Templates := "SrcType := Int" } EQ_Contact(in1 := "BUFFER".PROCESS, in2 := 210)
      wire#w2
      Contact( "RECIPE DB"."RINSE-2_SELECT" )
      { S7_Templates := "time_type := Time" } "IEC_Timer_0_DB_25".TON(pt := T#5s, et =>)
      Move(in := 300, out1 => "BUFFER".PROCESS)
   END_RUNG
   RUNG wire#w2
      I_Contact( "RECIPE DB"."RINSE-2_SELECT" )
      Move(in := 380, out1 => "BUFFER".PROCESS)
   END_RUNG
   RUNG wire#w1
      { S7_Templates := "SrcType := Int" } EQ_Contact(in1 := "BUFFER".PROCESS, in2 := 300)
      Contact( "CYCLE_POPUP"."RINSE-2_START_YES" )
      Move(in := 310, out1 => "BUFFER".PROCESS)
   END_RUNG
   RUNG wire#w1
      { S7_Templates := "SrcType := Int" } EQ_Contact(in1 := "BUFFER".PROCESS, in2 := 300)
      Contact( "CYCLE_POPUP"."RINSE-2_START_NO" )
      Move(in := 380, out1 => "BUFFER".PROCESS)
   END_RUNG
   // the same network as SCL:
   #_w1 := "AlwaysTRUE" AND ("BUFFER".PROCESS = 210);
   "IEC_Timer_0_DB_25".TON(IN := #_w1 AND "RECIPE DB"."RINSE-2_SELECT", PT := T#5s);
   IF "IEC_Timer_0_DB_25".Q THEN "BUFFER".PROCESS := 300; END_IF;
   IF #_w1 AND NOT "RECIPE DB"."RINSE-2_SELECT" THEN "BUFFER".PROCESS := 380; END_IF;
   IF "AlwaysTRUE" AND ("BUFFER".PROCESS = 300) AND "CYCLE_POPUP"."RINSE-2_START_YES" THEN
       "BUFFER".PROCESS := 310;
   END_IF;
   IF "AlwaysTRUE" AND ("BUFFER".PROCESS = 300) AND "CYCLE_POPUP"."RINSE-2_START_NO" THEN
       "BUFFER".PROCESS := 380;
   END_IF;
END_REGION

REGION Network 31: RINSE-2_SWT_LEVEL_CHECK (PBFV-18,17)
   RUNG wire#powerrail
      Contact( "AlwaysTRUE" )
      { S7_Templates := "SrcType := Int" } EQ_Contact(in1 := "BUFFER"."MODE SELECTION", in2 := 1)
      { S7_Templates := "SrcType := Int" } EQ_Contact(in1 := "BUFFER".PROCESS, in2 := 310)
      Contact( "IN".SWT_HL )
      Move(in := 320, out1 => "BUFFER".PROCESS)
   END_RUNG
   // the same network as SCL:
   IF "AlwaysTRUE" AND ("BUFFER"."MODE SELECTION" = 1) AND ("BUFFER".PROCESS = 310) AND "IN".SWT_HL THEN
       "BUFFER".PROCESS := 320;
   END_IF;
END_REGION

REGION Network 32: RINSE-2_TEMP_CHECK_(PBFV-1,PBFV-17,PZDV-1,F-PUMP,PBFV-3,PBFV-4,PBFV-8,CIP-IN)
   RUNG wire#powerrail
      Contact( "AlwaysTRUE" )
      { S7_Templates := "SrcType := Int" } EQ_Contact(in1 := "BUFFER"."MODE SELECTION", in2 := 1)
      { S7_Templates := "SrcType := Int" } EQ_Contact(in1 := "BUFFER".PROCESS, in2 := 320)
      { S7_Templates := "SrcType := Real" } GE_Contact(in1 := "SCALE_DB_TT".PV_VALUE, in2 := "SET_PARAMETERS"."RINSE-2_TEMPERATURE_SET")
      { S7_Templates := "time_type := Time" } "IEC_Timer_0_DB_6".TON(pt := T#5S, et =>)
      Move(in := 330, out1 => "BUFFER".PROCESS)
   END_RUNG
   // the same network as SCL:
   "IEC_Timer_0_DB_6".TON(IN := "AlwaysTRUE" AND ("BUFFER"."MODE SELECTION" = 1) AND ("BUFFER".PROCESS = 320) AND ("SCALE_DB_TT".PV_VALUE >= "SET_PARAMETERS"."RINSE-2_TEMPERATURE_SET"),
                          PT := T#5S);
   IF "IEC_Timer_0_DB_6".Q THEN "BUFFER".PROCESS := 330; END_IF;
END_REGION

REGION Network 33: RINSE-2_CLEANING_TIME_(PBFV-1,PBFV-17,PZDV-1,F-PUMP,PBFV-3,PBFV-4,PBFV-8,CIP-IN)
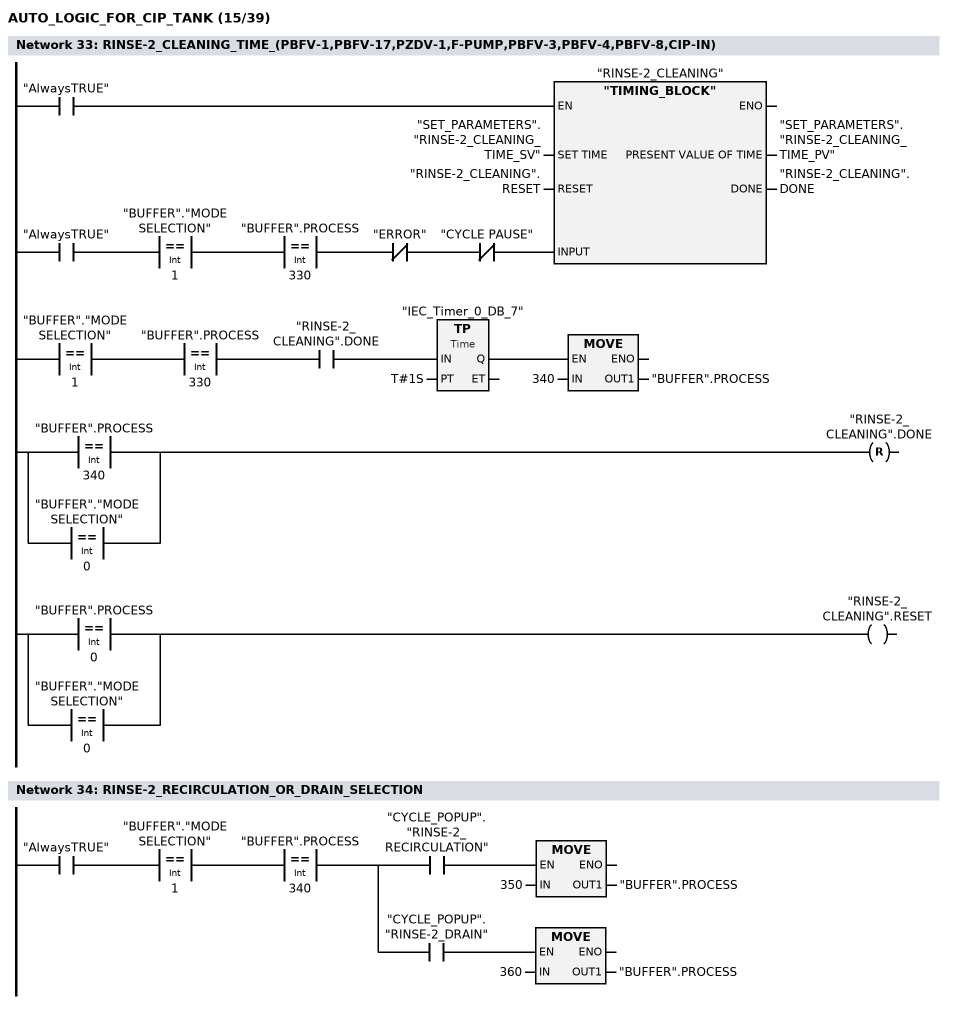
   RUNG wire#powerrail
      Contact( "AlwaysTRUE" )
      "RINSE-2_CLEANING"(INPUT := wire#w1, "SET TIME" := "SET_PARAMETERS"."RINSE-2_CLEANING_TIME_SV", RESET := "RINSE-2_CLEANING".RESET, "PRESENT VALUE OF TIME" => "SET_PARAMETERS"."RINSE-2_CLEANING_TIME_PV", DONE => "RINSE-2_CLEANING".DONE)
   END_RUNG
   RUNG wire#powerrail
      Contact( "AlwaysTRUE" )
      { S7_Templates := "SrcType := Int" } EQ_Contact(in1 := "BUFFER"."MODE SELECTION", in2 := 1)
      { S7_Templates := "SrcType := Int" } EQ_Contact(in1 := "BUFFER".PROCESS, in2 := 330)
      I_Contact( "ERROR" )
      I_Contact( "CYCLE PAUSE" )
   END_RUNG wire#w1
   RUNG wire#powerrail
      { S7_Templates := "SrcType := Int" } EQ_Contact(in1 := "BUFFER"."MODE SELECTION", in2 := 1)
      { S7_Templates := "SrcType := Int" } EQ_Contact(in1 := "BUFFER".PROCESS, in2 := 330)
      Contact( "RINSE-2_CLEANING".DONE )
      { S7_Templates := "time_type := Time" } "IEC_Timer_0_DB_7".TP(pt := T#1S, et =>)
      Move(in := 340, out1 => "BUFFER".PROCESS)
   END_RUNG
   RUNG wire#powerrail
      { S7_Templates := "SrcType := Int" } EQ_Contact(in1 := "BUFFER".PROCESS, in2 := 340)
      wire#w2
      R_Coil( "RINSE-2_CLEANING".DONE )
   END_RUNG
   RUNG wire#powerrail
      { S7_Templates := "SrcType := Int" } EQ_Contact(in1 := "BUFFER"."MODE SELECTION", in2 := 0)
   END_RUNG wire#w2
   RUNG wire#powerrail
      { S7_Templates := "SrcType := Int" } EQ_Contact(in1 := "BUFFER".PROCESS, in2 := 0)
      wire#w3
      Coil( "RINSE-2_CLEANING".RESET )
   END_RUNG
   RUNG wire#powerrail
      { S7_Templates := "SrcType := Int" } EQ_Contact(in1 := "BUFFER"."MODE SELECTION", in2 := 0)
   END_RUNG wire#w3
   // the same network as SCL:
   IF "AlwaysTRUE" THEN
       "RINSE-2_CLEANING"("SET TIME" := "SET_PARAMETERS"."RINSE-2_CLEANING_TIME_SV",   // "TIMING_BLOCK"
                          RESET := "RINSE-2_CLEANING".RESET,
                          INPUT := "AlwaysTRUE" AND ("BUFFER"."MODE SELECTION" = 1) AND ("BUFFER".PROCESS = 330) AND NOT "ERROR" AND NOT "CYCLE PAUSE",
                          "PRESENT VALUE OF TIME" => "SET_PARAMETERS"."RINSE-2_CLEANING_TIME_PV",
                          DONE => "RINSE-2_CLEANING".DONE);
   END_IF;
   "IEC_Timer_0_DB_7".TP(IN := ("BUFFER"."MODE SELECTION" = 1) AND ("BUFFER".PROCESS = 330) AND "RINSE-2_CLEANING".DONE,
                         PT := T#1S);
   IF "IEC_Timer_0_DB_7".Q THEN "BUFFER".PROCESS := 340; END_IF;
   IF ("BUFFER".PROCESS = 340) OR ("BUFFER"."MODE SELECTION" = 0) THEN
       "RINSE-2_CLEANING".DONE := FALSE;
   END_IF;
   "RINSE-2_CLEANING".RESET := ("BUFFER".PROCESS = 0) OR ("BUFFER"."MODE SELECTION" = 0);
END_REGION

REGION Network 34: RINSE-2_RECIRCULATION_OR_DRAIN_SELECTION
   RUNG wire#powerrail
      Contact( "AlwaysTRUE" )
      { S7_Templates := "SrcType := Int" } EQ_Contact(in1 := "BUFFER"."MODE SELECTION", in2 := 1)
      { S7_Templates := "SrcType := Int" } EQ_Contact(in1 := "BUFFER".PROCESS, in2 := 340)
      wire#w1
      Contact( "CYCLE_POPUP"."RINSE-2_RECIRCULATION" )
      Move(in := 350, out1 => "BUFFER".PROCESS)
   END_RUNG
   RUNG wire#w1
      Contact( "CYCLE_POPUP"."RINSE-2_DRAIN" )
      Move(in := 360, out1 => "BUFFER".PROCESS)
   END_RUNG
   // the same network as SCL:
   #_w1 := "AlwaysTRUE" AND ("BUFFER"."MODE SELECTION" = 1) AND ("BUFFER".PROCESS = 340);
   IF #_w1 AND "CYCLE_POPUP"."RINSE-2_RECIRCULATION" THEN "BUFFER".PROCESS := 350; END_IF;
   IF #_w1 AND "CYCLE_POPUP"."RINSE-2_DRAIN" THEN "BUFFER".PROCESS := 360; END_IF;
END_REGION

REGION Network 35: RINSE-2_RECIRCULATION_TIME_(CIP-OUT,R-PUMP,PBFV-6,PBFV-8,CIP-IN)
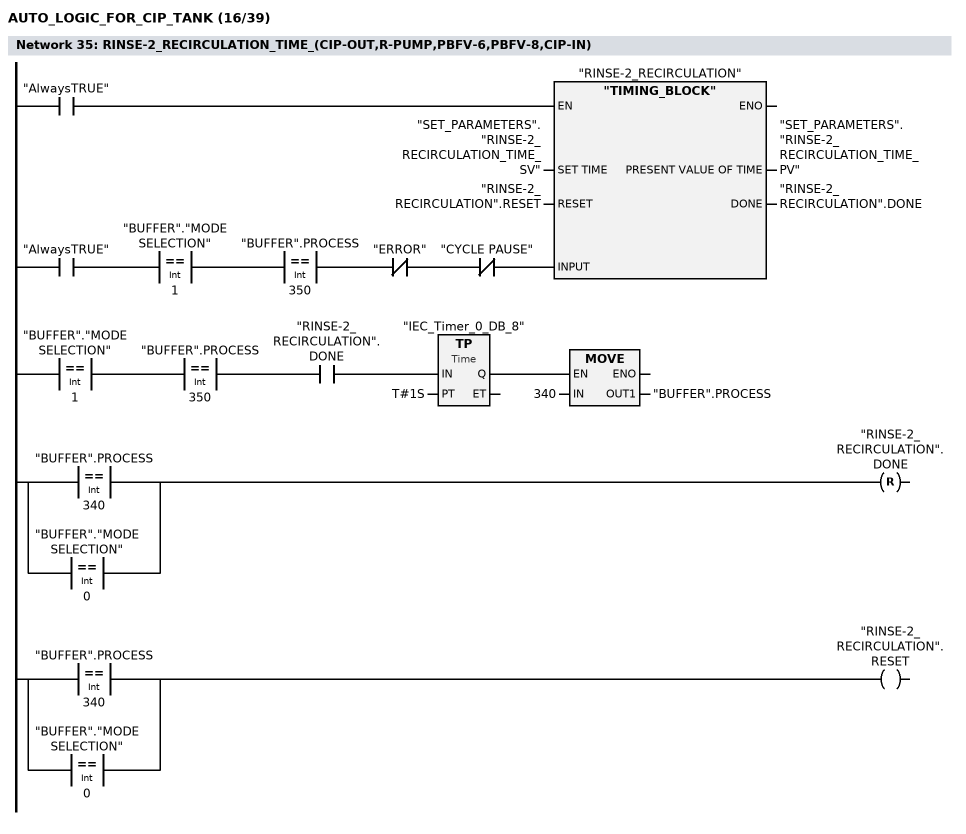
   RUNG wire#powerrail
      Contact( "AlwaysTRUE" )
      "RINSE-2_RECIRCULATION"(INPUT := wire#w1, "SET TIME" := "SET_PARAMETERS"."RINSE-2_RECIRCULATION_TIME_SV", RESET := "RINSE-2_RECIRCULATION".RESET, "PRESENT VALUE OF TIME" => "SET_PARAMETERS"."RINSE-2_RECIRCULATION_TIME_PV", DONE => "RINSE-2_RECIRCULATION".DONE)
   END_RUNG
   RUNG wire#powerrail
      Contact( "AlwaysTRUE" )
      { S7_Templates := "SrcType := Int" } EQ_Contact(in1 := "BUFFER"."MODE SELECTION", in2 := 1)
      { S7_Templates := "SrcType := Int" } EQ_Contact(in1 := "BUFFER".PROCESS, in2 := 350)
      I_Contact( "ERROR" )
      I_Contact( "CYCLE PAUSE" )
   END_RUNG wire#w1
   RUNG wire#powerrail
      { S7_Templates := "SrcType := Int" } EQ_Contact(in1 := "BUFFER"."MODE SELECTION", in2 := 1)
      { S7_Templates := "SrcType := Int" } EQ_Contact(in1 := "BUFFER".PROCESS, in2 := 350)
      Contact( "RINSE-2_RECIRCULATION".DONE )
      { S7_Templates := "time_type := Time" } "IEC_Timer_0_DB_8".TP(pt := T#1S, et =>)
      Move(in := 340, out1 => "BUFFER".PROCESS)
   END_RUNG
   RUNG wire#powerrail
      { S7_Templates := "SrcType := Int" } EQ_Contact(in1 := "BUFFER".PROCESS, in2 := 340)
      wire#w2
      R_Coil( "RINSE-2_RECIRCULATION".DONE )
   END_RUNG
   RUNG wire#powerrail
      { S7_Templates := "SrcType := Int" } EQ_Contact(in1 := "BUFFER"."MODE SELECTION", in2 := 0)
   END_RUNG wire#w2
   RUNG wire#powerrail
      { S7_Templates := "SrcType := Int" } EQ_Contact(in1 := "BUFFER".PROCESS, in2 := 340)
      wire#w3
      Coil( "RINSE-2_RECIRCULATION".RESET )
   END_RUNG
   RUNG wire#powerrail
      { S7_Templates := "SrcType := Int" } EQ_Contact(in1 := "BUFFER"."MODE SELECTION", in2 := 0)
   END_RUNG wire#w3
   // the same network as SCL:
   IF "AlwaysTRUE" THEN
       "RINSE-2_RECIRCULATION"("SET TIME" := "SET_PARAMETERS"."RINSE-2_RECIRCULATION_TIME_SV",   // "TIMING_BLOCK"
                               RESET := "RINSE-2_RECIRCULATION".RESET,
                               INPUT := "AlwaysTRUE" AND ("BUFFER"."MODE SELECTION" = 1) AND ("BUFFER".PROCESS = 350) AND NOT "ERROR" AND NOT "CYCLE PAUSE",
                               "PRESENT VALUE OF TIME" => "SET_PARAMETERS"."RINSE-2_RECIRCULATION_TIME_PV",
                               DONE => "RINSE-2_RECIRCULATION".DONE);
   END_IF;
   "IEC_Timer_0_DB_8".TP(IN := ("BUFFER"."MODE SELECTION" = 1) AND ("BUFFER".PROCESS = 350) AND "RINSE-2_RECIRCULATION".DONE,
                         PT := T#1S);
   IF "IEC_Timer_0_DB_8".Q THEN "BUFFER".PROCESS := 340; END_IF;
   IF ("BUFFER".PROCESS = 340) OR ("BUFFER"."MODE SELECTION" = 0) THEN
       "RINSE-2_RECIRCULATION".DONE := FALSE;
   END_IF;
   "RINSE-2_RECIRCULATION".RESET := ("BUFFER".PROCESS = 340) OR ("BUFFER"."MODE SELECTION" = 0);
END_REGION

REGION Network 36: RINSE-2_DRAIN_TIME_(CIP-OUT,R_PUMP,PBFV-11)
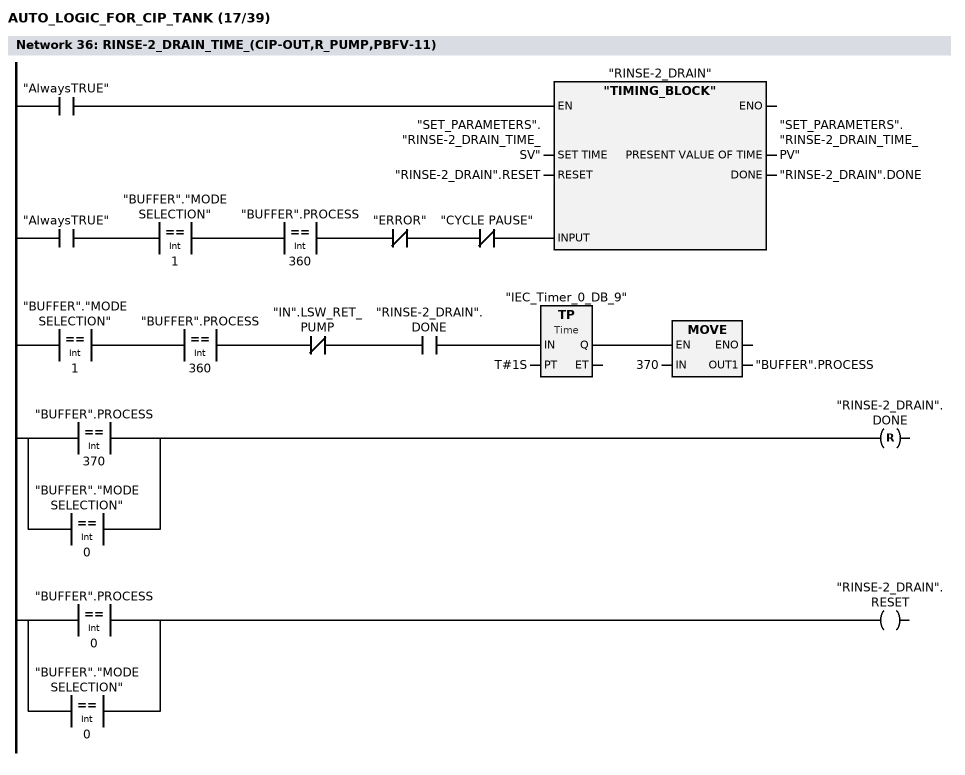
   RUNG wire#powerrail
      Contact( "AlwaysTRUE" )
      "RINSE-2_DRAIN"(INPUT := wire#w1, "SET TIME" := "SET_PARAMETERS"."RINSE-2_DRAIN_TIME_SV", RESET := "RINSE-2_DRAIN".RESET, "PRESENT VALUE OF TIME" => "SET_PARAMETERS"."RINSE-2_DRAIN_TIME_PV", DONE => "RINSE-2_DRAIN".DONE)
   END_RUNG
   RUNG wire#powerrail
      Contact( "AlwaysTRUE" )
      { S7_Templates := "SrcType := Int" } EQ_Contact(in1 := "BUFFER"."MODE SELECTION", in2 := 1)
      { S7_Templates := "SrcType := Int" } EQ_Contact(in1 := "BUFFER".PROCESS, in2 := 360)
      I_Contact( "ERROR" )
      I_Contact( "CYCLE PAUSE" )
   END_RUNG wire#w1
   RUNG wire#powerrail
      { S7_Templates := "SrcType := Int" } EQ_Contact(in1 := "BUFFER"."MODE SELECTION", in2 := 1)
      { S7_Templates := "SrcType := Int" } EQ_Contact(in1 := "BUFFER".PROCESS, in2 := 360)
      I_Contact( "IN".LSW_RET_PUMP )
      Contact( "RINSE-2_DRAIN".DONE )
      { S7_Templates := "time_type := Time" } "IEC_Timer_0_DB_9".TP(pt := T#1S, et =>)
      Move(in := 370, out1 => "BUFFER".PROCESS)
   END_RUNG
   RUNG wire#powerrail
      { S7_Templates := "SrcType := Int" } EQ_Contact(in1 := "BUFFER".PROCESS, in2 := 370)
      wire#w2
      R_Coil( "RINSE-2_DRAIN".DONE )
   END_RUNG
   RUNG wire#powerrail
      { S7_Templates := "SrcType := Int" } EQ_Contact(in1 := "BUFFER"."MODE SELECTION", in2 := 0)
   END_RUNG wire#w2
   RUNG wire#powerrail
      { S7_Templates := "SrcType := Int" } EQ_Contact(in1 := "BUFFER".PROCESS, in2 := 0)
      wire#w3
      Coil( "RINSE-2_DRAIN".RESET )
   END_RUNG
   RUNG wire#powerrail
      { S7_Templates := "SrcType := Int" } EQ_Contact(in1 := "BUFFER"."MODE SELECTION", in2 := 0)
   END_RUNG wire#w3
   // the same network as SCL:
   IF "AlwaysTRUE" THEN
       "RINSE-2_DRAIN"("SET TIME" := "SET_PARAMETERS"."RINSE-2_DRAIN_TIME_SV",   // "TIMING_BLOCK"
                       RESET := "RINSE-2_DRAIN".RESET,
                       INPUT := "AlwaysTRUE" AND ("BUFFER"."MODE SELECTION" = 1) AND ("BUFFER".PROCESS = 360) AND NOT "ERROR" AND NOT "CYCLE PAUSE",
                       "PRESENT VALUE OF TIME" => "SET_PARAMETERS"."RINSE-2_DRAIN_TIME_PV",
                       DONE => "RINSE-2_DRAIN".DONE);
   END_IF;
   "IEC_Timer_0_DB_9".TP(IN := ("BUFFER"."MODE SELECTION" = 1) AND ("BUFFER".PROCESS = 360) AND NOT "IN".LSW_RET_PUMP AND "RINSE-2_DRAIN".DONE,
                         PT := T#1S);
   IF "IEC_Timer_0_DB_9".Q THEN "BUFFER".PROCESS := 370; END_IF;
   IF ("BUFFER".PROCESS = 370) OR ("BUFFER"."MODE SELECTION" = 0) THEN "RINSE-2_DRAIN".DONE := FALSE; END_IF;
   "RINSE-2_DRAIN".RESET := ("BUFFER".PROCESS = 0) OR ("BUFFER"."MODE SELECTION" = 0);
END_REGION

REGION Network 37: RINSE-2_PUMP_CHASING_TIME_(PBFV-12,PBFV13)
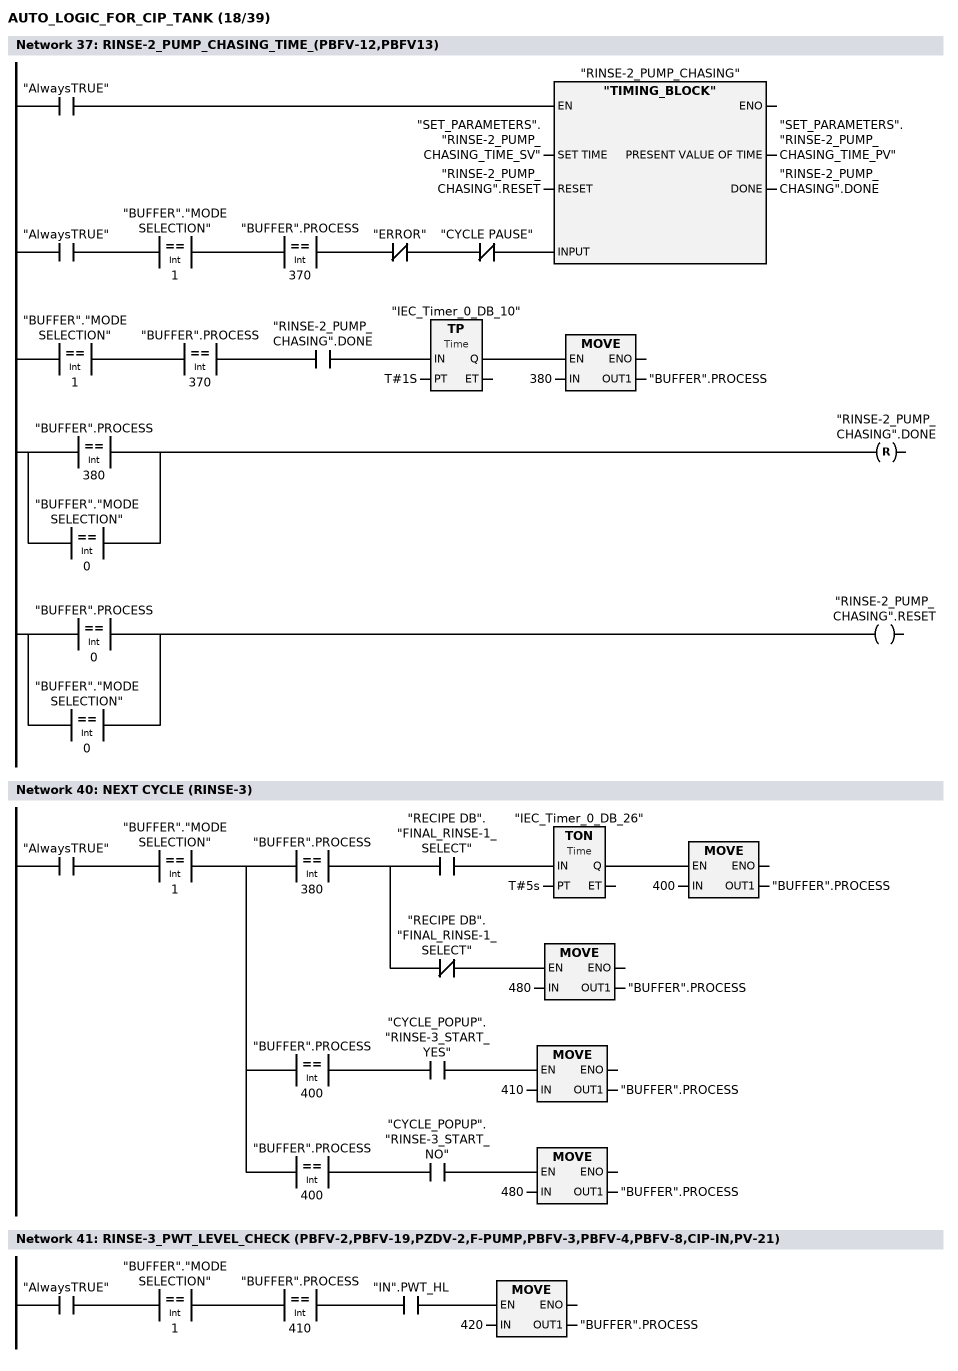
   RUNG wire#powerrail
      Contact( "AlwaysTRUE" )
      "RINSE-2_PUMP_CHASING"(INPUT := wire#w1, "SET TIME" := "SET_PARAMETERS"."RINSE-2_PUMP_CHASING_TIME_SV", RESET := "RINSE-2_PUMP_CHASING".RESET, "PRESENT VALUE OF TIME" => "SET_PARAMETERS"."RINSE-2_PUMP_CHASING_TIME_PV", DONE => "RINSE-2_PUMP_CHASING".DONE)
   END_RUNG
   RUNG wire#powerrail
      Contact( "AlwaysTRUE" )
      { S7_Templates := "SrcType := Int" } EQ_Contact(in1 := "BUFFER"."MODE SELECTION", in2 := 1)
      { S7_Templates := "SrcType := Int" } EQ_Contact(in1 := "BUFFER".PROCESS, in2 := 370)
      I_Contact( "ERROR" )
      I_Contact( "CYCLE PAUSE" )
   END_RUNG wire#w1
   RUNG wire#powerrail
      { S7_Templates := "SrcType := Int" } EQ_Contact(in1 := "BUFFER"."MODE SELECTION", in2 := 1)
      { S7_Templates := "SrcType := Int" } EQ_Contact(in1 := "BUFFER".PROCESS, in2 := 370)
      Contact( "RINSE-2_PUMP_CHASING".DONE )
      { S7_Templates := "time_type := Time" } "IEC_Timer_0_DB_10".TP(pt := T#1S, et =>)
      Move(in := 380, out1 => "BUFFER".PROCESS)
   END_RUNG
   RUNG wire#powerrail
      { S7_Templates := "SrcType := Int" } EQ_Contact(in1 := "BUFFER".PROCESS, in2 := 380)
      wire#w2
      R_Coil( "RINSE-2_PUMP_CHASING".DONE )
   END_RUNG
   RUNG wire#powerrail
      { S7_Templates := "SrcType := Int" } EQ_Contact(in1 := "BUFFER"."MODE SELECTION", in2 := 0)
   END_RUNG wire#w2
   RUNG wire#powerrail
      { S7_Templates := "SrcType := Int" } EQ_Contact(in1 := "BUFFER".PROCESS, in2 := 0)
      wire#w3
      Coil( "RINSE-2_PUMP_CHASING".RESET )
   END_RUNG
   RUNG wire#powerrail
      { S7_Templates := "SrcType := Int" } EQ_Contact(in1 := "BUFFER"."MODE SELECTION", in2 := 0)
   END_RUNG wire#w3
   // the same network as SCL:
   IF "AlwaysTRUE" THEN
       "RINSE-2_PUMP_CHASING"("SET TIME" := "SET_PARAMETERS"."RINSE-2_PUMP_CHASING_TIME_SV",   // "TIMING_BLOCK"
                              RESET := "RINSE-2_PUMP_CHASING".RESET,
                              INPUT := "AlwaysTRUE" AND ("BUFFER"."MODE SELECTION" = 1) AND ("BUFFER".PROCESS = 370) AND NOT "ERROR" AND NOT "CYCLE PAUSE",
                              "PRESENT VALUE OF TIME" => "SET_PARAMETERS"."RINSE-2_PUMP_CHASING_TIME_PV",
                              DONE => "RINSE-2_PUMP_CHASING".DONE);
   END_IF;
   "IEC_Timer_0_DB_10".TP(IN := ("BUFFER"."MODE SELECTION" = 1) AND ("BUFFER".PROCESS = 370) AND "RINSE-2_PUMP_CHASING".DONE,
                          PT := T#1S);
   IF "IEC_Timer_0_DB_10".Q THEN "BUFFER".PROCESS := 380; END_IF;
   IF ("BUFFER".PROCESS = 380) OR ("BUFFER"."MODE SELECTION" = 0) THEN
       "RINSE-2_PUMP_CHASING".DONE := FALSE;
   END_IF;
   "RINSE-2_PUMP_CHASING".RESET := ("BUFFER".PROCESS = 0) OR ("BUFFER"."MODE SELECTION" = 0);
END_REGION

REGION Network 40: NEXT CYCLE (RINSE-3)
   RUNG wire#powerrail
      Contact( "AlwaysTRUE" )
      { S7_Templates := "SrcType := Int" } EQ_Contact(in1 := "BUFFER"."MODE SELECTION", in2 := 1)
      wire#w1
      { S7_Templates := "SrcType := Int" } EQ_Contact(in1 := "BUFFER".PROCESS, in2 := 380)
      wire#w2
      Contact( "RECIPE DB"."FINAL_RINSE-1_SELECT" )
      { S7_Templates := "time_type := Time" } "IEC_Timer_0_DB_26".TON(pt := T#5s, et =>)
      Move(in := 400, out1 => "BUFFER".PROCESS)
   END_RUNG
   RUNG wire#w2
      I_Contact( "RECIPE DB"."FINAL_RINSE-1_SELECT" )
      Move(in := 480, out1 => "BUFFER".PROCESS)
   END_RUNG
   RUNG wire#w1
      { S7_Templates := "SrcType := Int" } EQ_Contact(in1 := "BUFFER".PROCESS, in2 := 400)
      Contact( "CYCLE_POPUP"."RINSE-3_START_YES" )
      Move(in := 410, out1 => "BUFFER".PROCESS)
   END_RUNG
   RUNG wire#w1
      { S7_Templates := "SrcType := Int" } EQ_Contact(in1 := "BUFFER".PROCESS, in2 := 400)
      Contact( "CYCLE_POPUP"."RINSE-3_START_NO" )
      Move(in := 480, out1 => "BUFFER".PROCESS)
   END_RUNG
   // the same network as SCL:
   #_w1 := "AlwaysTRUE" AND ("BUFFER"."MODE SELECTION" = 1);
   #_w2 := #_w1 AND ("BUFFER".PROCESS = 380);
   "IEC_Timer_0_DB_26".TON(IN := #_w2 AND "RECIPE DB"."FINAL_RINSE-1_SELECT", PT := T#5s);
   IF "IEC_Timer_0_DB_26".Q THEN "BUFFER".PROCESS := 400; END_IF;
   IF #_w2 AND NOT "RECIPE DB"."FINAL_RINSE-1_SELECT" THEN "BUFFER".PROCESS := 480; END_IF;
   IF #_w1 AND ("BUFFER".PROCESS = 400) AND "CYCLE_POPUP"."RINSE-3_START_YES" THEN
       "BUFFER".PROCESS := 410;
   END_IF;
   IF #_w1 AND ("BUFFER".PROCESS = 400) AND "CYCLE_POPUP"."RINSE-3_START_NO" THEN
       "BUFFER".PROCESS := 480;
   END_IF;
END_REGION

REGION Network 41: RINSE-3_PWT_LEVEL_CHECK (PBFV-2,PBFV-19,PZDV-2,F-PUMP,PBFV-3,PBFV-4,PBFV-8,CIP-IN,PV-21)
   RUNG wire#powerrail
      Contact( "AlwaysTRUE" )
      { S7_Templates := "SrcType := Int" } EQ_Contact(in1 := "BUFFER"."MODE SELECTION", in2 := 1)
      { S7_Templates := "SrcType := Int" } EQ_Contact(in1 := "BUFFER".PROCESS, in2 := 410)
      Contact( "IN".PWT_HL )
      Move(in := 420, out1 => "BUFFER".PROCESS)
   END_RUNG
   // the same network as SCL:
   IF "AlwaysTRUE" AND ("BUFFER"."MODE SELECTION" = 1) AND ("BUFFER".PROCESS = 410) AND "IN".PWT_HL THEN
       "BUFFER".PROCESS := 420;
   END_IF;
END_REGION

REGION Network 42: RINSE-3_TEMP_CHECK _(PBFV-2,PBFV-19,PZDV-2,F-PUMP,PBFV-3,PBFV-4,PBFV-8,CIP-IN)
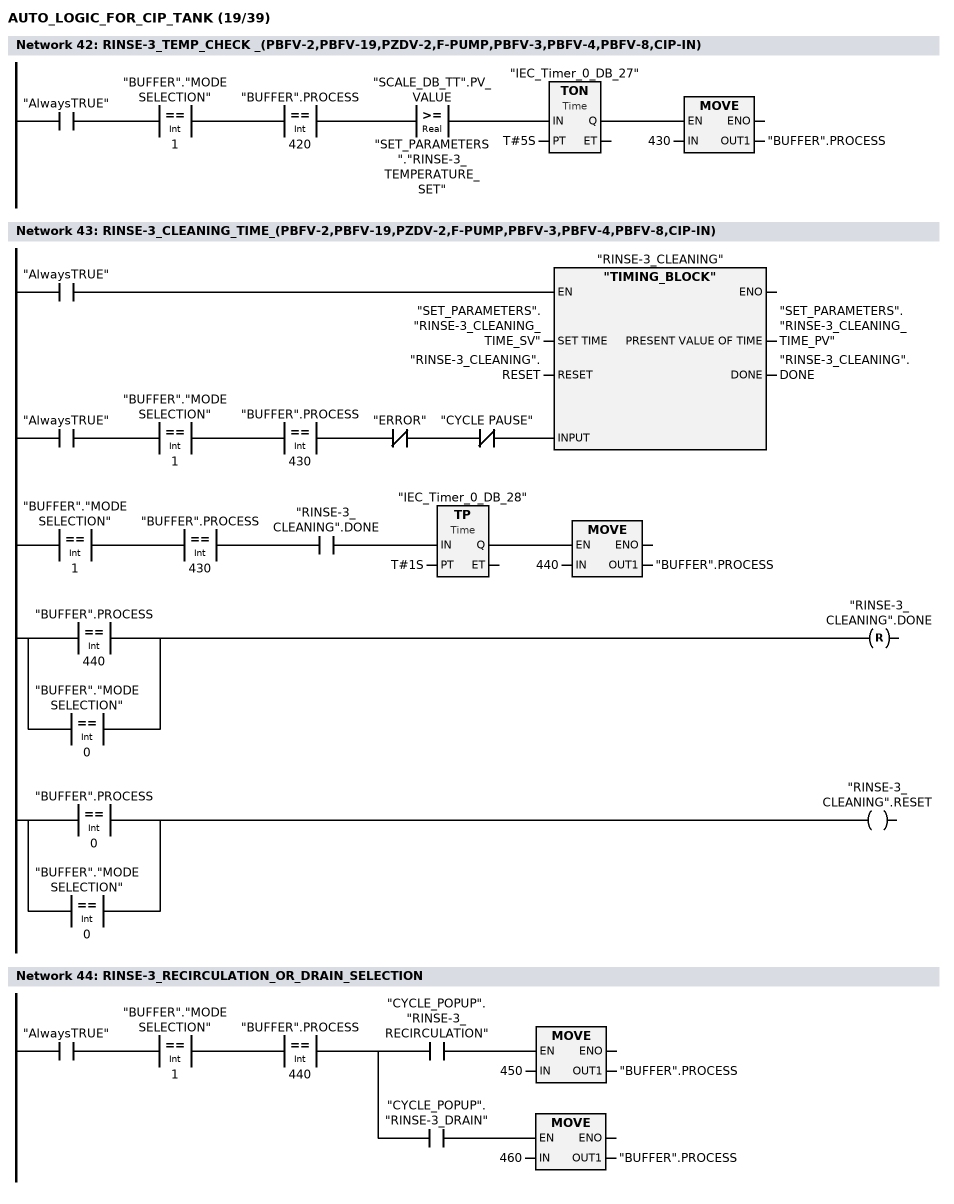
   RUNG wire#powerrail
      Contact( "AlwaysTRUE" )
      { S7_Templates := "SrcType := Int" } EQ_Contact(in1 := "BUFFER"."MODE SELECTION", in2 := 1)
      { S7_Templates := "SrcType := Int" } EQ_Contact(in1 := "BUFFER".PROCESS, in2 := 420)
      { S7_Templates := "SrcType := Real" } GE_Contact(in1 := "SCALE_DB_TT".PV_VALUE, in2 := "SET_PARAMETERS"."RINSE-3_TEMPERATURE_SET")
      { S7_Templates := "time_type := Time" } "IEC_Timer_0_DB_27".TON(pt := T#5S, et =>)
      Move(in := 430, out1 => "BUFFER".PROCESS)
   END_RUNG
   // the same network as SCL:
   "IEC_Timer_0_DB_27".TON(IN := "AlwaysTRUE" AND ("BUFFER"."MODE SELECTION" = 1) AND ("BUFFER".PROCESS = 420) AND ("SCALE_DB_TT".PV_VALUE >= "SET_PARAMETERS"."RINSE-3_TEMPERATURE_SET"),
                           PT := T#5S);
   IF "IEC_Timer_0_DB_27".Q THEN "BUFFER".PROCESS := 430; END_IF;
END_REGION

REGION Network 43: RINSE-3_CLEANING_TIME_(PBFV-2,PBFV-19,PZDV-2,F-PUMP,PBFV-3,PBFV-4,PBFV-8,CIP-IN)
   RUNG wire#powerrail
      Contact( "AlwaysTRUE" )
      "RINSE-3_CLEANING"(INPUT := wire#w1, "SET TIME" := "SET_PARAMETERS"."RINSE-3_CLEANING_TIME_SV", RESET := "RINSE-3_CLEANING".RESET, "PRESENT VALUE OF TIME" => "SET_PARAMETERS"."RINSE-3_CLEANING_TIME_PV", DONE => "RINSE-3_CLEANING".DONE)
   END_RUNG
   RUNG wire#powerrail
      Contact( "AlwaysTRUE" )
      { S7_Templates := "SrcType := Int" } EQ_Contact(in1 := "BUFFER"."MODE SELECTION", in2 := 1)
      { S7_Templates := "SrcType := Int" } EQ_Contact(in1 := "BUFFER".PROCESS, in2 := 430)
      I_Contact( "ERROR" )
      I_Contact( "CYCLE PAUSE" )
   END_RUNG wire#w1
   RUNG wire#powerrail
      { S7_Templates := "SrcType := Int" } EQ_Contact(in1 := "BUFFER"."MODE SELECTION", in2 := 1)
      { S7_Templates := "SrcType := Int" } EQ_Contact(in1 := "BUFFER".PROCESS, in2 := 430)
      Contact( "RINSE-3_CLEANING".DONE )
      { S7_Templates := "time_type := Time" } "IEC_Timer_0_DB_28".TP(pt := T#1S, et =>)
      Move(in := 440, out1 => "BUFFER".PROCESS)
   END_RUNG
   RUNG wire#powerrail
      { S7_Templates := "SrcType := Int" } EQ_Contact(in1 := "BUFFER".PROCESS, in2 := 440)
      wire#w2
      R_Coil( "RINSE-3_CLEANING".DONE )
   END_RUNG
   RUNG wire#powerrail
      { S7_Templates := "SrcType := Int" } EQ_Contact(in1 := "BUFFER"."MODE SELECTION", in2 := 0)
   END_RUNG wire#w2
   RUNG wire#powerrail
      { S7_Templates := "SrcType := Int" } EQ_Contact(in1 := "BUFFER".PROCESS, in2 := 0)
      wire#w3
      Coil( "RINSE-3_CLEANING".RESET )
   END_RUNG
   RUNG wire#powerrail
      { S7_Templates := "SrcType := Int" } EQ_Contact(in1 := "BUFFER"."MODE SELECTION", in2 := 0)
   END_RUNG wire#w3
   // the same network as SCL:
   IF "AlwaysTRUE" THEN
       "RINSE-3_CLEANING"("SET TIME" := "SET_PARAMETERS"."RINSE-3_CLEANING_TIME_SV",   // "TIMING_BLOCK"
                          RESET := "RINSE-3_CLEANING".RESET,
                          INPUT := "AlwaysTRUE" AND ("BUFFER"."MODE SELECTION" = 1) AND ("BUFFER".PROCESS = 430) AND NOT "ERROR" AND NOT "CYCLE PAUSE",
                          "PRESENT VALUE OF TIME" => "SET_PARAMETERS"."RINSE-3_CLEANING_TIME_PV",
                          DONE => "RINSE-3_CLEANING".DONE);
   END_IF;
   "IEC_Timer_0_DB_28".TP(IN := ("BUFFER"."MODE SELECTION" = 1) AND ("BUFFER".PROCESS = 430) AND "RINSE-3_CLEANING".DONE,
                          PT := T#1S);
   IF "IEC_Timer_0_DB_28".Q THEN "BUFFER".PROCESS := 440; END_IF;
   IF ("BUFFER".PROCESS = 440) OR ("BUFFER"."MODE SELECTION" = 0) THEN
       "RINSE-3_CLEANING".DONE := FALSE;
   END_IF;
   "RINSE-3_CLEANING".RESET := ("BUFFER".PROCESS = 0) OR ("BUFFER"."MODE SELECTION" = 0);
END_REGION

REGION Network 44: RINSE-3_RECIRCULATION_OR_DRAIN_SELECTION
   RUNG wire#powerrail
      Contact( "AlwaysTRUE" )
      { S7_Templates := "SrcType := Int" } EQ_Contact(in1 := "BUFFER"."MODE SELECTION", in2 := 1)
      { S7_Templates := "SrcType := Int" } EQ_Contact(in1 := "BUFFER".PROCESS, in2 := 440)
      wire#w1
      Contact( "CYCLE_POPUP"."RINSE-3_RECIRCULATION" )
      Move(in := 450, out1 => "BUFFER".PROCESS)
   END_RUNG
   RUNG wire#w1
      Contact( "CYCLE_POPUP"."RINSE-3_DRAIN" )
      Move(in := 460, out1 => "BUFFER".PROCESS)
   END_RUNG
   // the same network as SCL:
   #_w1 := "AlwaysTRUE" AND ("BUFFER"."MODE SELECTION" = 1) AND ("BUFFER".PROCESS = 440);
   IF #_w1 AND "CYCLE_POPUP"."RINSE-3_RECIRCULATION" THEN "BUFFER".PROCESS := 450; END_IF;
   IF #_w1 AND "CYCLE_POPUP"."RINSE-3_DRAIN" THEN "BUFFER".PROCESS := 460; END_IF;
END_REGION

REGION Network 45: RINSE-3_RECIRCULATION_TIME_(CIP-OUT,R-PUMP,PBFV-6,PBFV-8,CIP-IN)
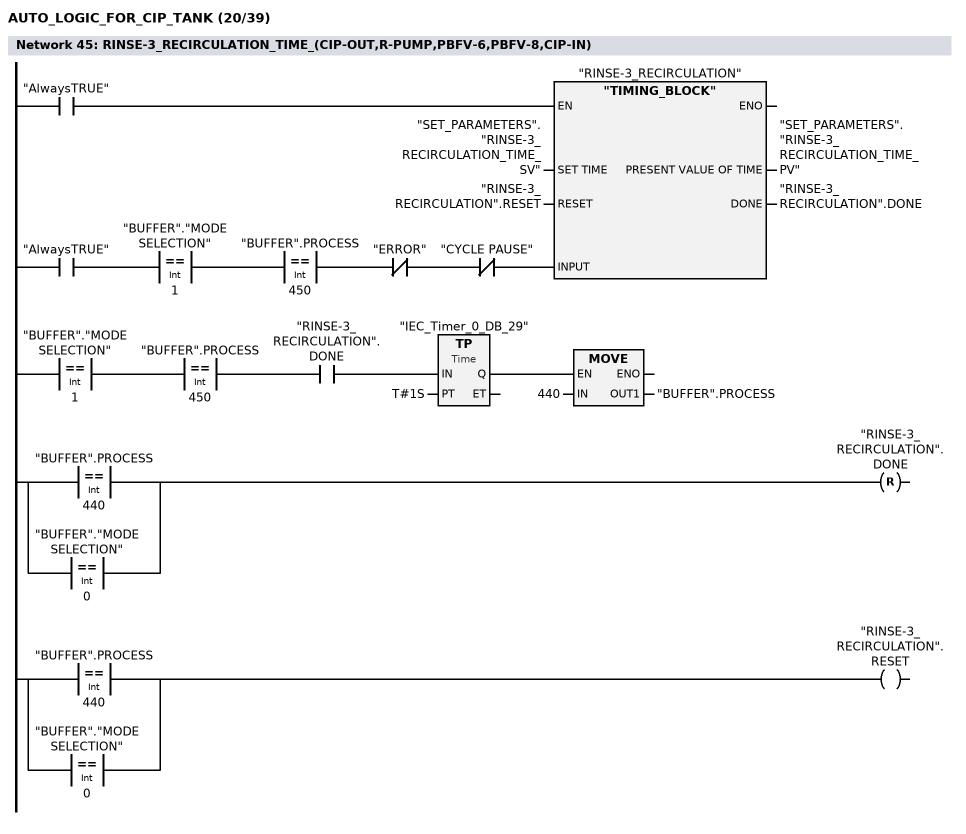
   RUNG wire#powerrail
      Contact( "AlwaysTRUE" )
      "RINSE-3_RECIRCULATION"(INPUT := wire#w1, "SET TIME" := "SET_PARAMETERS"."RINSE-3_RECIRCULATION_TIME_SV", RESET := "RINSE-3_RECIRCULATION".RESET, "PRESENT VALUE OF TIME" => "SET_PARAMETERS"."RINSE-3_RECIRCULATION_TIME_PV", DONE => "RINSE-3_RECIRCULATION".DONE)
   END_RUNG
   RUNG wire#powerrail
      Contact( "AlwaysTRUE" )
      { S7_Templates := "SrcType := Int" } EQ_Contact(in1 := "BUFFER"."MODE SELECTION", in2 := 1)
      { S7_Templates := "SrcType := Int" } EQ_Contact(in1 := "BUFFER".PROCESS, in2 := 450)
      I_Contact( "ERROR" )
      I_Contact( "CYCLE PAUSE" )
   END_RUNG wire#w1
   RUNG wire#powerrail
      { S7_Templates := "SrcType := Int" } EQ_Contact(in1 := "BUFFER"."MODE SELECTION", in2 := 1)
      { S7_Templates := "SrcType := Int" } EQ_Contact(in1 := "BUFFER".PROCESS, in2 := 450)
      Contact( "RINSE-3_RECIRCULATION".DONE )
      { S7_Templates := "time_type := Time" } "IEC_Timer_0_DB_29".TP(pt := T#1S, et =>)
      Move(in := 440, out1 => "BUFFER".PROCESS)
   END_RUNG
   RUNG wire#powerrail
      { S7_Templates := "SrcType := Int" } EQ_Contact(in1 := "BUFFER".PROCESS, in2 := 440)
      wire#w2
      R_Coil( "RINSE-3_RECIRCULATION".DONE )
   END_RUNG
   RUNG wire#powerrail
      { S7_Templates := "SrcType := Int" } EQ_Contact(in1 := "BUFFER"."MODE SELECTION", in2 := 0)
   END_RUNG wire#w2
   RUNG wire#powerrail
      { S7_Templates := "SrcType := Int" } EQ_Contact(in1 := "BUFFER".PROCESS, in2 := 440)
      wire#w3
      Coil( "RINSE-3_RECIRCULATION".RESET )
   END_RUNG
   RUNG wire#powerrail
      { S7_Templates := "SrcType := Int" } EQ_Contact(in1 := "BUFFER"."MODE SELECTION", in2 := 0)
   END_RUNG wire#w3
   // the same network as SCL:
   IF "AlwaysTRUE" THEN
       "RINSE-3_RECIRCULATION"("SET TIME" := "SET_PARAMETERS"."RINSE-3_RECIRCULATION_TIME_SV",   // "TIMING_BLOCK"
                               RESET := "RINSE-3_RECIRCULATION".RESET,
                               INPUT := "AlwaysTRUE" AND ("BUFFER"."MODE SELECTION" = 1) AND ("BUFFER".PROCESS = 450) AND NOT "ERROR" AND NOT "CYCLE PAUSE",
                               "PRESENT VALUE OF TIME" => "SET_PARAMETERS"."RINSE-3_RECIRCULATION_TIME_PV",
                               DONE => "RINSE-3_RECIRCULATION".DONE);
   END_IF;
   "IEC_Timer_0_DB_29".TP(IN := ("BUFFER"."MODE SELECTION" = 1) AND ("BUFFER".PROCESS = 450) AND "RINSE-3_RECIRCULATION".DONE,
                          PT := T#1S);
   IF "IEC_Timer_0_DB_29".Q THEN "BUFFER".PROCESS := 440; END_IF;
   IF ("BUFFER".PROCESS = 440) OR ("BUFFER"."MODE SELECTION" = 0) THEN
       "RINSE-3_RECIRCULATION".DONE := FALSE;
   END_IF;
   "RINSE-3_RECIRCULATION".RESET := ("BUFFER".PROCESS = 440) OR ("BUFFER"."MODE SELECTION" = 0);
END_REGION

REGION Network 46: RINSE-3_DRAIN_TIME_(CIP-OUT,R_PUMP,PBFV-11)
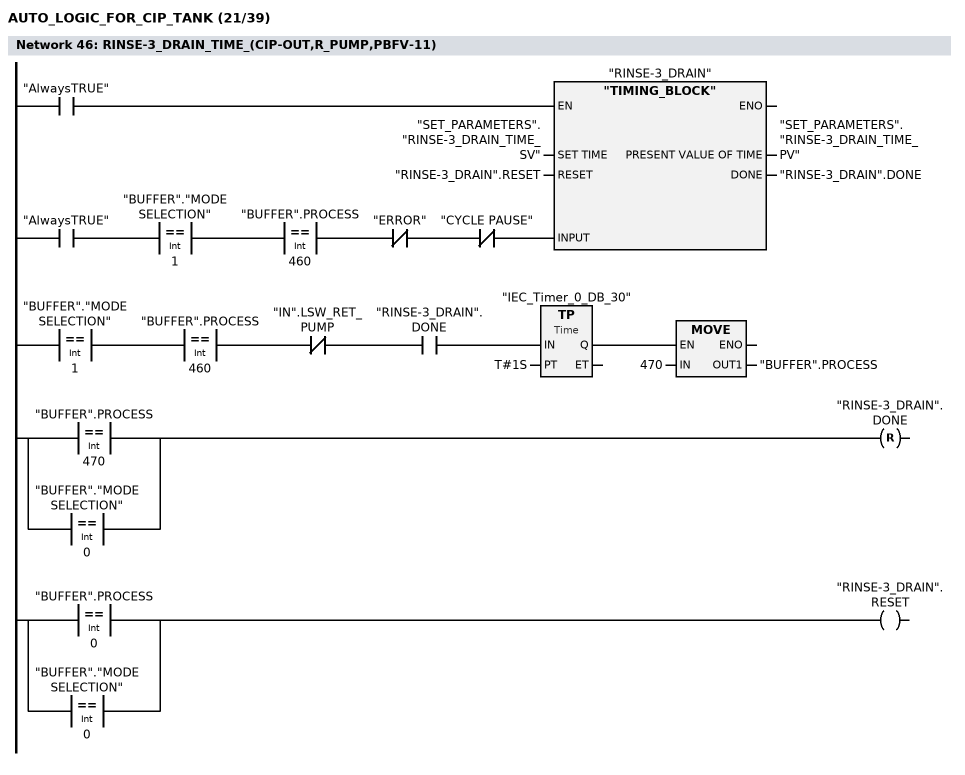
   RUNG wire#powerrail
      Contact( "AlwaysTRUE" )
      "RINSE-3_DRAIN"(INPUT := wire#w1, "SET TIME" := "SET_PARAMETERS"."RINSE-3_DRAIN_TIME_SV", RESET := "RINSE-3_DRAIN".RESET, "PRESENT VALUE OF TIME" => "SET_PARAMETERS"."RINSE-3_DRAIN_TIME_PV", DONE => "RINSE-3_DRAIN".DONE)
   END_RUNG
   RUNG wire#powerrail
      Contact( "AlwaysTRUE" )
      { S7_Templates := "SrcType := Int" } EQ_Contact(in1 := "BUFFER"."MODE SELECTION", in2 := 1)
      { S7_Templates := "SrcType := Int" } EQ_Contact(in1 := "BUFFER".PROCESS, in2 := 460)
      I_Contact( "ERROR" )
      I_Contact( "CYCLE PAUSE" )
   END_RUNG wire#w1
   RUNG wire#powerrail
      { S7_Templates := "SrcType := Int" } EQ_Contact(in1 := "BUFFER"."MODE SELECTION", in2 := 1)
      { S7_Templates := "SrcType := Int" } EQ_Contact(in1 := "BUFFER".PROCESS, in2 := 460)
      I_Contact( "IN".LSW_RET_PUMP )
      Contact( "RINSE-3_DRAIN".DONE )
      { S7_Templates := "time_type := Time" } "IEC_Timer_0_DB_30".TP(pt := T#1S, et =>)
      Move(in := 470, out1 => "BUFFER".PROCESS)
   END_RUNG
   RUNG wire#powerrail
      { S7_Templates := "SrcType := Int" } EQ_Contact(in1 := "BUFFER".PROCESS, in2 := 470)
      wire#w2
      R_Coil( "RINSE-3_DRAIN".DONE )
   END_RUNG
   RUNG wire#powerrail
      { S7_Templates := "SrcType := Int" } EQ_Contact(in1 := "BUFFER"."MODE SELECTION", in2 := 0)
   END_RUNG wire#w2
   RUNG wire#powerrail
      { S7_Templates := "SrcType := Int" } EQ_Contact(in1 := "BUFFER".PROCESS, in2 := 0)
      wire#w3
      Coil( "RINSE-3_DRAIN".RESET )
   END_RUNG
   RUNG wire#powerrail
      { S7_Templates := "SrcType := Int" } EQ_Contact(in1 := "BUFFER"."MODE SELECTION", in2 := 0)
   END_RUNG wire#w3
   // the same network as SCL:
   IF "AlwaysTRUE" THEN
       "RINSE-3_DRAIN"("SET TIME" := "SET_PARAMETERS"."RINSE-3_DRAIN_TIME_SV",   // "TIMING_BLOCK"
                       RESET := "RINSE-3_DRAIN".RESET,
                       INPUT := "AlwaysTRUE" AND ("BUFFER"."MODE SELECTION" = 1) AND ("BUFFER".PROCESS = 460) AND NOT "ERROR" AND NOT "CYCLE PAUSE",
                       "PRESENT VALUE OF TIME" => "SET_PARAMETERS"."RINSE-3_DRAIN_TIME_PV",
                       DONE => "RINSE-3_DRAIN".DONE);
   END_IF;
   "IEC_Timer_0_DB_30".TP(IN := ("BUFFER"."MODE SELECTION" = 1) AND ("BUFFER".PROCESS = 460) AND NOT "IN".LSW_RET_PUMP AND "RINSE-3_DRAIN".DONE,
                          PT := T#1S);
   IF "IEC_Timer_0_DB_30".Q THEN "BUFFER".PROCESS := 470; END_IF;
   IF ("BUFFER".PROCESS = 470) OR ("BUFFER"."MODE SELECTION" = 0) THEN "RINSE-3_DRAIN".DONE := FALSE; END_IF;
   "RINSE-3_DRAIN".RESET := ("BUFFER".PROCESS = 0) OR ("BUFFER"."MODE SELECTION" = 0);
END_REGION

REGION Network 47: RINSE-3_PUMP_CHASING_TIME_(PBFV-12,PBFV13)
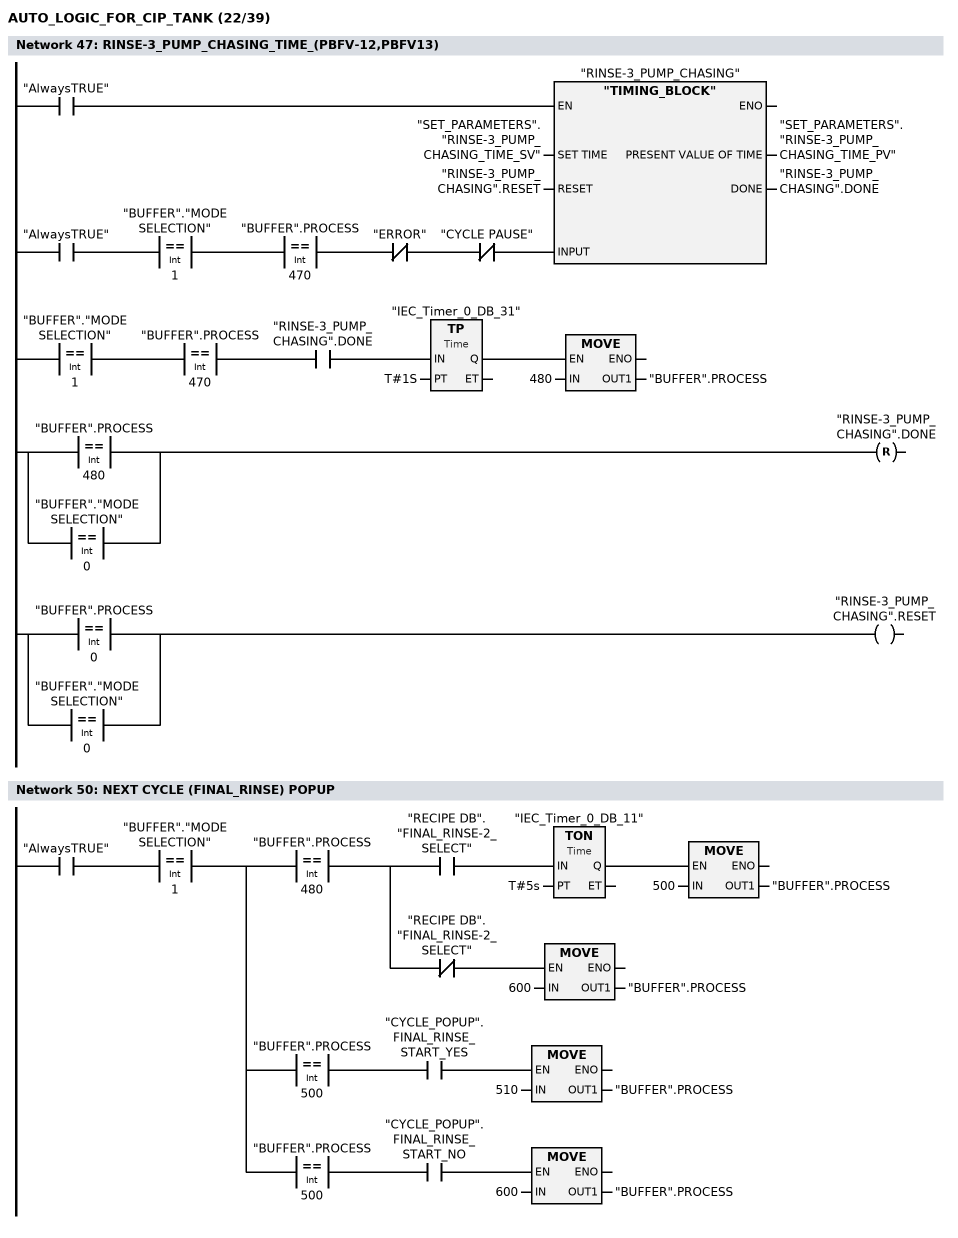
   RUNG wire#powerrail
      Contact( "AlwaysTRUE" )
      "RINSE-3_PUMP_CHASING"(INPUT := wire#w1, "SET TIME" := "SET_PARAMETERS"."RINSE-3_PUMP_CHASING_TIME_SV", RESET := "RINSE-3_PUMP_CHASING".RESET, "PRESENT VALUE OF TIME" => "SET_PARAMETERS"."RINSE-3_PUMP_CHASING_TIME_PV", DONE => "RINSE-3_PUMP_CHASING".DONE)
   END_RUNG
   RUNG wire#powerrail
      Contact( "AlwaysTRUE" )
      { S7_Templates := "SrcType := Int" } EQ_Contact(in1 := "BUFFER"."MODE SELECTION", in2 := 1)
      { S7_Templates := "SrcType := Int" } EQ_Contact(in1 := "BUFFER".PROCESS, in2 := 470)
      I_Contact( "ERROR" )
      I_Contact( "CYCLE PAUSE" )
   END_RUNG wire#w1
   RUNG wire#powerrail
      { S7_Templates := "SrcType := Int" } EQ_Contact(in1 := "BUFFER"."MODE SELECTION", in2 := 1)
      { S7_Templates := "SrcType := Int" } EQ_Contact(in1 := "BUFFER".PROCESS, in2 := 470)
      Contact( "RINSE-3_PUMP_CHASING".DONE )
      { S7_Templates := "time_type := Time" } "IEC_Timer_0_DB_31".TP(pt := T#1S, et =>)
      Move(in := 480, out1 => "BUFFER".PROCESS)
   END_RUNG
   RUNG wire#powerrail
      { S7_Templates := "SrcType := Int" } EQ_Contact(in1 := "BUFFER".PROCESS, in2 := 480)
      wire#w2
      R_Coil( "RINSE-3_PUMP_CHASING".DONE )
   END_RUNG
   RUNG wire#powerrail
      { S7_Templates := "SrcType := Int" } EQ_Contact(in1 := "BUFFER"."MODE SELECTION", in2 := 0)
   END_RUNG wire#w2
   RUNG wire#powerrail
      { S7_Templates := "SrcType := Int" } EQ_Contact(in1 := "BUFFER".PROCESS, in2 := 0)
      wire#w3
      Coil( "RINSE-3_PUMP_CHASING".RESET )
   END_RUNG
   RUNG wire#powerrail
      { S7_Templates := "SrcType := Int" } EQ_Contact(in1 := "BUFFER"."MODE SELECTION", in2 := 0)
   END_RUNG wire#w3
   // the same network as SCL:
   IF "AlwaysTRUE" THEN
       "RINSE-3_PUMP_CHASING"("SET TIME" := "SET_PARAMETERS"."RINSE-3_PUMP_CHASING_TIME_SV",   // "TIMING_BLOCK"
                              RESET := "RINSE-3_PUMP_CHASING".RESET,
                              INPUT := "AlwaysTRUE" AND ("BUFFER"."MODE SELECTION" = 1) AND ("BUFFER".PROCESS = 470) AND NOT "ERROR" AND NOT "CYCLE PAUSE",
                              "PRESENT VALUE OF TIME" => "SET_PARAMETERS"."RINSE-3_PUMP_CHASING_TIME_PV",
                              DONE => "RINSE-3_PUMP_CHASING".DONE);
   END_IF;
   "IEC_Timer_0_DB_31".TP(IN := ("BUFFER"."MODE SELECTION" = 1) AND ("BUFFER".PROCESS = 470) AND "RINSE-3_PUMP_CHASING".DONE,
                          PT := T#1S);
   IF "IEC_Timer_0_DB_31".Q THEN "BUFFER".PROCESS := 480; END_IF;
   IF ("BUFFER".PROCESS = 480) OR ("BUFFER"."MODE SELECTION" = 0) THEN
       "RINSE-3_PUMP_CHASING".DONE := FALSE;
   END_IF;
   "RINSE-3_PUMP_CHASING".RESET := ("BUFFER".PROCESS = 0) OR ("BUFFER"."MODE SELECTION" = 0);
END_REGION

REGION Network 50: NEXT CYCLE (FINAL_RINSE) POPUP
   RUNG wire#powerrail
      Contact( "AlwaysTRUE" )
      { S7_Templates := "SrcType := Int" } EQ_Contact(in1 := "BUFFER"."MODE SELECTION", in2 := 1)
      wire#w1
      { S7_Templates := "SrcType := Int" } EQ_Contact(in1 := "BUFFER".PROCESS, in2 := 480)
      wire#w2
      Contact( "RECIPE DB"."FINAL_RINSE-2_SELECT" )
      { S7_Templates := "time_type := Time" } "IEC_Timer_0_DB_11".TON(pt := T#5s, et =>)
      Move(in := 500, out1 => "BUFFER".PROCESS)
   END_RUNG
   RUNG wire#w2
      I_Contact( "RECIPE DB"."FINAL_RINSE-2_SELECT" )
      Move(in := 600, out1 => "BUFFER".PROCESS)
   END_RUNG
   RUNG wire#w1
      { S7_Templates := "SrcType := Int" } EQ_Contact(in1 := "BUFFER".PROCESS, in2 := 500)
      Contact( "CYCLE_POPUP".FINAL_RINSE_START_YES )
      Move(in := 510, out1 => "BUFFER".PROCESS)
   END_RUNG
   RUNG wire#w1
      { S7_Templates := "SrcType := Int" } EQ_Contact(in1 := "BUFFER".PROCESS, in2 := 500)
      Contact( "CYCLE_POPUP".FINAL_RINSE_START_NO )
      Move(in := 600, out1 => "BUFFER".PROCESS)
   END_RUNG
   // the same network as SCL:
   #_w1 := "AlwaysTRUE" AND ("BUFFER"."MODE SELECTION" = 1);
   #_w2 := #_w1 AND ("BUFFER".PROCESS = 480);
   "IEC_Timer_0_DB_11".TON(IN := #_w2 AND "RECIPE DB"."FINAL_RINSE-2_SELECT", PT := T#5s);
   IF "IEC_Timer_0_DB_11".Q THEN "BUFFER".PROCESS := 500; END_IF;
   IF #_w2 AND NOT "RECIPE DB"."FINAL_RINSE-2_SELECT" THEN "BUFFER".PROCESS := 600; END_IF;
   IF #_w1 AND ("BUFFER".PROCESS = 500) AND "CYCLE_POPUP".FINAL_RINSE_START_YES THEN
       "BUFFER".PROCESS := 510;
   END_IF;
   IF #_w1 AND ("BUFFER".PROCESS = 500) AND "CYCLE_POPUP".FINAL_RINSE_START_NO THEN
       "BUFFER".PROCESS := 600;
   END_IF;
END_REGION

REGION Network 51: PWT_LEVEL_CHECK
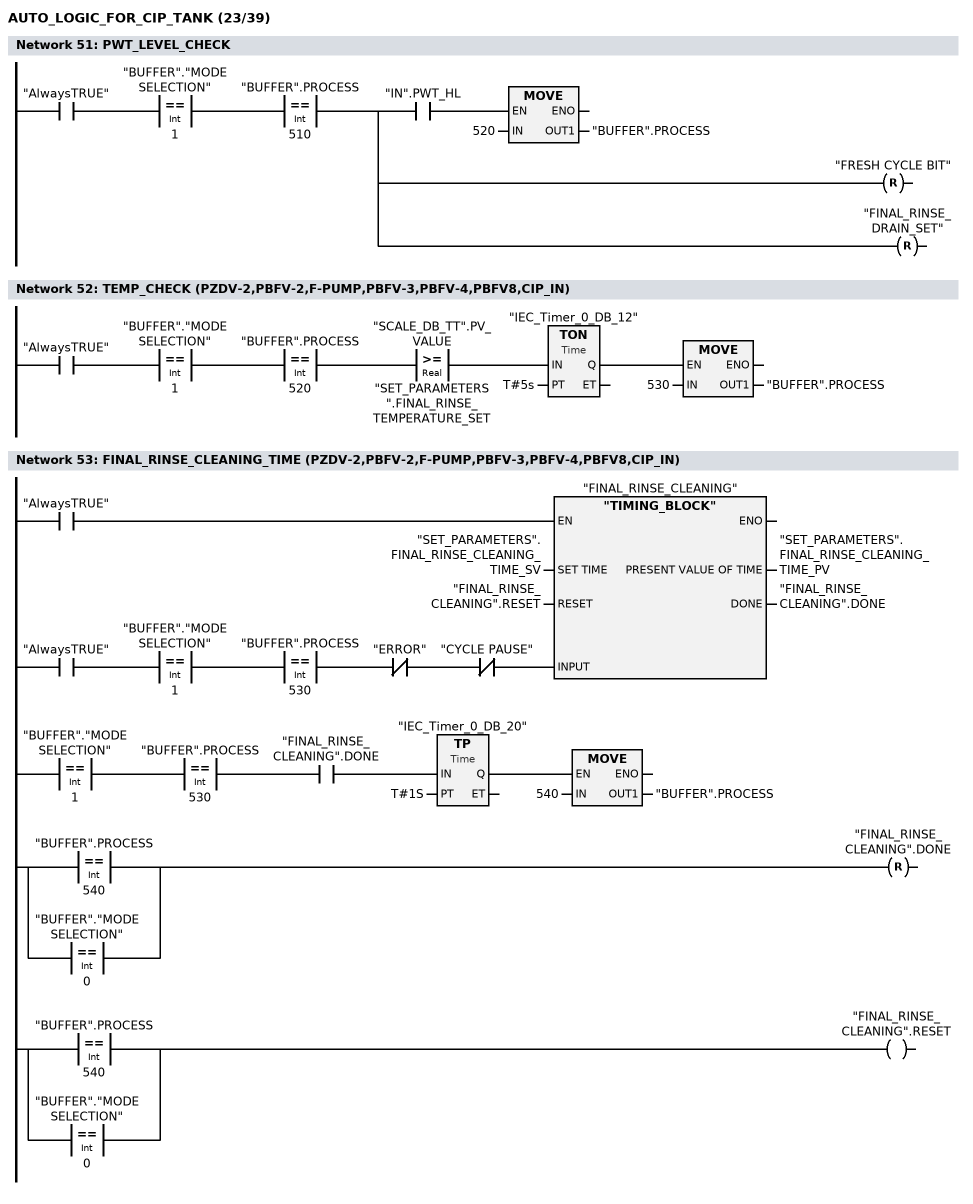
   RUNG wire#powerrail
      Contact( "AlwaysTRUE" )
      { S7_Templates := "SrcType := Int" } EQ_Contact(in1 := "BUFFER"."MODE SELECTION", in2 := 1)
      { S7_Templates := "SrcType := Int" } EQ_Contact(in1 := "BUFFER".PROCESS, in2 := 510)
      wire#w1
      Contact( "IN".PWT_HL )
      Move(in := 520, out1 => "BUFFER".PROCESS)
   END_RUNG
   RUNG wire#w1
      R_Coil( "FRESH CYCLE BIT" )
   END_RUNG
   RUNG wire#w1
      R_Coil( "FINAL_RINSE_DRAIN_SET" )
   END_RUNG
   // the same network as SCL:
   #_w1 := "AlwaysTRUE" AND ("BUFFER"."MODE SELECTION" = 1) AND ("BUFFER".PROCESS = 510);
   IF #_w1 AND "IN".PWT_HL THEN "BUFFER".PROCESS := 520; END_IF;
   IF #_w1 THEN
       "FRESH CYCLE BIT" := FALSE;
       "FINAL_RINSE_DRAIN_SET" := FALSE;
   END_IF;
END_REGION

REGION Network 52: TEMP_CHECK (PZDV-2,PBFV-2,F-PUMP,PBFV-3,PBFV-4,PBFV8,CIP_IN)
   RUNG wire#powerrail
      Contact( "AlwaysTRUE" )
      { S7_Templates := "SrcType := Int" } EQ_Contact(in1 := "BUFFER"."MODE SELECTION", in2 := 1)
      { S7_Templates := "SrcType := Int" } EQ_Contact(in1 := "BUFFER".PROCESS, in2 := 520)
      { S7_Templates := "SrcType := Real" } GE_Contact(in1 := "SCALE_DB_TT".PV_VALUE, in2 := "SET_PARAMETERS".FINAL_RINSE_TEMPERATURE_SET)
      { S7_Templates := "time_type := Time" } "IEC_Timer_0_DB_12".TON(pt := T#5s, et =>)
      Move(in := 530, out1 => "BUFFER".PROCESS)
   END_RUNG
   // the same network as SCL:
   "IEC_Timer_0_DB_12".TON(IN := "AlwaysTRUE" AND ("BUFFER"."MODE SELECTION" = 1) AND ("BUFFER".PROCESS = 520) AND ("SCALE_DB_TT".PV_VALUE >= "SET_PARAMETERS".FINAL_RINSE_TEMPERATURE_SET),
                           PT := T#5s);
   IF "IEC_Timer_0_DB_12".Q THEN "BUFFER".PROCESS := 530; END_IF;
END_REGION

REGION Network 53: FINAL_RINSE_CLEANING_TIME (PZDV-2,PBFV-2,F-PUMP,PBFV-3,PBFV-4,PBFV8,CIP_IN)
   RUNG wire#powerrail
      Contact( "AlwaysTRUE" )
      "FINAL_RINSE_CLEANING"(INPUT := wire#w1, "SET TIME" := "SET_PARAMETERS".FINAL_RINSE_CLEANING_TIME_SV, RESET := "FINAL_RINSE_CLEANING".RESET, "PRESENT VALUE OF TIME" => "SET_PARAMETERS".FINAL_RINSE_CLEANING_TIME_PV, DONE => "FINAL_RINSE_CLEANING".DONE)
   END_RUNG
   RUNG wire#powerrail
      Contact( "AlwaysTRUE" )
      { S7_Templates := "SrcType := Int" } EQ_Contact(in1 := "BUFFER"."MODE SELECTION", in2 := 1)
      { S7_Templates := "SrcType := Int" } EQ_Contact(in1 := "BUFFER".PROCESS, in2 := 530)
      I_Contact( "ERROR" )
      I_Contact( "CYCLE PAUSE" )
   END_RUNG wire#w1
   RUNG wire#powerrail
      { S7_Templates := "SrcType := Int" } EQ_Contact(in1 := "BUFFER"."MODE SELECTION", in2 := 1)
      { S7_Templates := "SrcType := Int" } EQ_Contact(in1 := "BUFFER".PROCESS, in2 := 530)
      Contact( "FINAL_RINSE_CLEANING".DONE )
      { S7_Templates := "time_type := Time" } "IEC_Timer_0_DB_20".TP(pt := T#1S, et =>)
      Move(in := 540, out1 => "BUFFER".PROCESS)
   END_RUNG
   RUNG wire#powerrail
      { S7_Templates := "SrcType := Int" } EQ_Contact(in1 := "BUFFER".PROCESS, in2 := 540)
      wire#w2
      R_Coil( "FINAL_RINSE_CLEANING".DONE )
   END_RUNG
   RUNG wire#powerrail
      { S7_Templates := "SrcType := Int" } EQ_Contact(in1 := "BUFFER"."MODE SELECTION", in2 := 0)
   END_RUNG wire#w2
   RUNG wire#powerrail
      { S7_Templates := "SrcType := Int" } EQ_Contact(in1 := "BUFFER".PROCESS, in2 := 540)
      wire#w3
      Coil( "FINAL_RINSE_CLEANING".RESET )
   END_RUNG
   RUNG wire#powerrail
      { S7_Templates := "SrcType := Int" } EQ_Contact(in1 := "BUFFER"."MODE SELECTION", in2 := 0)
   END_RUNG wire#w3
   // the same network as SCL:
   IF "AlwaysTRUE" THEN
       "FINAL_RINSE_CLEANING"("SET TIME" := "SET_PARAMETERS".FINAL_RINSE_CLEANING_TIME_SV,   // "TIMING_BLOCK"
                              RESET := "FINAL_RINSE_CLEANING".RESET,
                              INPUT := "AlwaysTRUE" AND ("BUFFER"."MODE SELECTION" = 1) AND ("BUFFER".PROCESS = 530) AND NOT "ERROR" AND NOT "CYCLE PAUSE",
                              "PRESENT VALUE OF TIME" => "SET_PARAMETERS".FINAL_RINSE_CLEANING_TIME_PV,
                              DONE => "FINAL_RINSE_CLEANING".DONE);
   END_IF;
   "IEC_Timer_0_DB_20".TP(IN := ("BUFFER"."MODE SELECTION" = 1) AND ("BUFFER".PROCESS = 530) AND "FINAL_RINSE_CLEANING".DONE,
                          PT := T#1S);
   IF "IEC_Timer_0_DB_20".Q THEN "BUFFER".PROCESS := 540; END_IF;
   IF ("BUFFER".PROCESS = 540) OR ("BUFFER"."MODE SELECTION" = 0) THEN
       "FINAL_RINSE_CLEANING".DONE := FALSE;
   END_IF;
   "FINAL_RINSE_CLEANING".RESET := ("BUFFER".PROCESS = 540) OR ("BUFFER"."MODE SELECTION" = 0);
END_REGION

REGION Network 54: CONDUCTIVITY ACHIEVED OR NOT ACHIEVED BIT SET
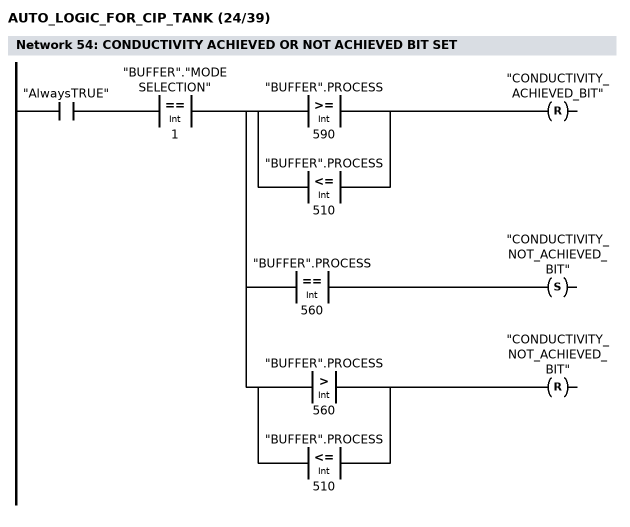
   RUNG wire#powerrail
      Contact( "AlwaysTRUE" )
      { S7_Templates := "SrcType := Int" } EQ_Contact(in1 := "BUFFER"."MODE SELECTION", in2 := 1)
      wire#w1
      { S7_Templates := "SrcType := Int" } GE_Contact(in1 := "BUFFER".PROCESS, in2 := 590)
      wire#w2
      R_Coil( "CONDUCTIVITY_ACHIEVED_BIT" )
   END_RUNG
   RUNG wire#w1
      { S7_Templates := "SrcType := Int" } LE_Contact(in1 := "BUFFER".PROCESS, in2 := 510)
   END_RUNG wire#w2
   RUNG wire#w1
      { S7_Templates := "SrcType := Int" } EQ_Contact(in1 := "BUFFER".PROCESS, in2 := 560)
      S_Coil( "CONDUCTIVITY_NOT_ACHIEVED_BIT" )
   END_RUNG
   RUNG wire#w1
      { S7_Templates := "SrcType := Int" } GT_Contact(in1 := "BUFFER".PROCESS, in2 := 560)
      wire#w3
      R_Coil( "CONDUCTIVITY_NOT_ACHIEVED_BIT" )
   END_RUNG
   RUNG wire#w1
      { S7_Templates := "SrcType := Int" } LE_Contact(in1 := "BUFFER".PROCESS, in2 := 510)
   END_RUNG wire#w3
   // the same network as SCL:
   #_w1 := "AlwaysTRUE" AND ("BUFFER"."MODE SELECTION" = 1);
   IF #_w1 AND (("BUFFER".PROCESS >= 590) OR ("BUFFER".PROCESS <= 510)) THEN
       "CONDUCTIVITY_ACHIEVED_BIT" := FALSE;
   END_IF;
   IF #_w1 AND ("BUFFER".PROCESS = 560) THEN "CONDUCTIVITY_NOT_ACHIEVED_BIT" := TRUE; END_IF;
   IF #_w1 AND (("BUFFER".PROCESS > 560) OR ("BUFFER".PROCESS <= 510)) THEN
       "CONDUCTIVITY_NOT_ACHIEVED_BIT" := FALSE;
   END_IF;
END_REGION

REGION Network 55: FINAL_RINSE_CONDUCTIVITY CHECKING TIME
